LIN {X 0,Y 546.313,Z 765.202,A -85,B 0,C 180,E1 25447.625,E2 25447.625} C_VEL
LIN {X 0,Y 547.105,Z 747.49,A -85,B 0,C 180,E1 25445.835,E2 25445.835} C_VEL
LIN {X 0,Y 547.912,Z 730.024,A -85,B 0,C 180,E1 25444.317,E2 25444.317} C_VEL
LIN {X 0,Y 548.795,Z 710.07,A -85,B 0,C 180,E1 25442.846,E2 25442.846} C_VEL
LIN {X 0,Y 549.579,Z 691.702,A -85,B 0,C 180,E1 25441.708,E2 25441.708} C_VEL
LIN {X 0,Y 550.398,Z 670.915,A -85,B 0,C 180,E1 25440.628,E2 25440.628} C_VEL
LIN {X 0,Y 551.103,Z 650.987,A -85,B 0,C 180,E1 25439.802,E2 25439.802} C_VEL
LIN {X 0,Y 551.691,Z 629.673,A -85,B 0,C 180,E1 25439.106,E2 25439.106} C_VEL
LIN {X 0,Y 552.189,Z 607.333,A -85,B 0,C 180,E1 25438.596,E2 25438.596} C_VEL
LIN {X 0,Y 553.481,Z 453.484,A -85,B 0,C 180,E1 25436.326,E2 25436.326} C_VEL
LIN {X 0,Y 554.426,Z 320.88,A -85,B 0,C 180,E1 25434.346,E2 25434.346} C_VEL
LIN {X 0,Y 549.959,Z 305.52,A -85,B 0,C 180,E1 25433.742,E2 25433.742} C_VEL
LIN {X 0,Y 550.398,Z 290.694,A -85,B 0,C 180,E1 25431.989,E2 25431.989} C_VEL
LIN {X 0,Y 545.865,Z 277.355,A -85,B 0,C 180,E1 25429.964,E2 25429.964} C_VEL
LIN {X 0,Y 544.39,Z 272.482,A -85,B 0,C 180,E1 25429.174,E2 25429.174} C_VEL
LIN {X 0,Y 544.34,Z 272.43,A -85,B 0,C 180,E1 25426.028,E2 25426.028} C_VEL
LIN {X 0,Y 544.339,Z 272.424,A -85,B 0,C 180,E1 25422.562,E2 25422.562} C_VEL
LIN {X 0,Y 544.397,Z 272.403,A -85,B 0,C 180,E1 25419.358,E2 25419.358} C_VEL
LIN {X 0,Y 544.337,Z 272.425,A -85,B 0,C 180,E1 25416.081,E2 25416.081} C_VEL
LIN {X 0,Y 544.365,Z 272.425,A -85,B 0,C 180,E1 25412.733,E2 25412.733} C_VEL
LIN {X 0,Y 544.362,Z 272.42,A -85,B 0,C 180,E1 25409.609,E2 25409.609} C_VEL
LIN {X 0,Y 544.344,Z 272.417,A -85,B 0,C 180,E1 25406.274,E2 25406.274} C_VEL
LIN {X 0,Y 544.409,Z 272.422,A -85,B 0,C 180,E1 25403.029,E2 25403.029} C_VEL
LIN {X 0,Y 544.349,Z 272.415,A -85,B 0,C 180,E1 25399.753,E2 25399.753} C_VEL
LIN {X 0,Y 544.358,Z 272.418,A -85,B 0,C 180,E1 25396.321,E2 25396.321} C_VEL
LIN {X 0,Y 544.4,Z 272.421,A -85,B 0,C 180,E1 25393.056,E2 25393.056} C_VEL
LIN {X 0,Y 544.35,Z 272.418,A -85,B 0,C 180,E1 25389.729,E2 25389.729} C_VEL
LIN {X 0,Y 544.384,Z 272.422,A -85,B 0,C 180,E1 25386.433,E2 25386.433} C_VEL
LIN {X 0,Y 544.382,Z 272.416,A -85,B 0,C 180,E1 25383.159,E2 25383.159} C_VEL
LIN {X 0,Y 544.354,Z 272.423,A -85,B 0,C 180,E1 25379.79,E2 25379.79} C_VEL
LIN {X 0,Y 544.402,Z 272.411,A -85,B 0,C 180,E1 25376.525,E2 25376.525} C_VEL
LIN {X 0,Y 544.369,Z 272.425,A -85,B 0,C 180,E1 25373.249,E2 25373.249} C_VEL
LIN {X 0,Y 544.364,Z 272.413,A -85,B 0,C 180,E1 25369.844,E2 25369.844} C_VEL
LIN {X 0,Y 544.406,Z 272.418,A -85,B 0,C 180,E1 25366.512,E2 25366.512} C_VEL
LIN {X 0,Y 544.366,Z 272.417,A -85,B 0,C 180,E1 25363.24,E2 25363.24} C_VEL
LIN {X 0,Y 544.374,Z 272.42,A -85,B 0,C 180,E1 25359.8,E2 25359.8} C_VEL
LIN {X 0,Y 544.406,Z 272.424,A -85,B 0,C 180,E1 25356.513,E2 25356.513} C_VEL
LIN {X 0,Y 544.37,Z 272.424,A -85,B 0,C 180,E1 25353.139,E2 25353.139} C_VEL
LIN {X 0,Y 544.378,Z 272.421,A -85,B 0,C 180,E1 25349.663,E2 25349.663} C_VEL
LIN {X 0,Y 544.374,Z 272.425,A -85,B 0,C 180,E1 25349.04,E2 25349.04} C_VEL
LIN {X 0,Y 543.409,Z 272.55,A -85,B 0,C 180,E1 25348.229,E2 25348.229} C_VEL
LIN {X 0,Y 536.878,Z 273.358,A -85,B 0,C 180,E1 25345.892,E2 25345.892} C_VEL
LIN {X 0,Y 536.432,Z 273.411,A -85,B 0,C 180,E1 25345.358,E2 25345.358} C_VEL
LIN {X 0,Y 536.464,Z 273.409,A -85,B 0,C 180,E1 25342.033,E2 25342.033} C_VEL
LIN {X 0,Y 536.459,Z 273.413,A -85,B 0,C 180,E1 25338.574,E2 25338.574} C_VEL
LIN {X 0,Y 536.436,Z 273.411,A -85,B 0,C 180,E1 25335.207,E2 25335.207} C_VEL
LIN {X 0,Y 536.465,Z 273.408,A -85,B 0,C 180,E1 25331.797,E2 25331.797} C_VEL
LIN {X 0,Y 536.465,Z 273.414,A -85,B 0,C 180,E1 25328.311,E2 25328.311} C_VEL
LIN {X 0,Y 536.441,Z 273.412,A -85,B 0,C 180,E1 25324.903,E2 25324.903} C_VEL
LIN {X 0,Y 536.461,Z 273.407,A -85,B 0,C 180,E1 25321.456,E2 25321.456} C_VEL
LIN {X 0,Y 536.459,Z 273.411,A -85,B 0,C 180,E1 25318.013,E2 25318.013} C_VEL
LIN {X 0,Y 536.444,Z 273.411,A -85,B 0,C 180,E1 25314.676,E2 25314.676} C_VEL
LIN {X 0,Y 536.457,Z 273.407,A -85,B 0,C 180,E1 25311.197,E2 25311.197} C_VEL
LIN {X 0,Y 536.456,Z 273.411,A -85,B 0,C 180,E1 25307.747,E2 25307.747} C_VEL
LIN {X 0,Y 536.455,Z 273.415,A -85,B 0,C 180,E1 25304.352,E2 25304.352} C_VEL
LIN {X 0,Y 536.45,Z 273.41,A -85,B 0,C 180,E1 25300.85,E2 25300.85} C_VEL
LIN {X 0,Y 536.452,Z 273.41,A -85,B 0,C 180,E1 25297.45,E2 25297.45} C_VEL
LIN {X 0,Y 536.46,Z 273.414,A -85,B 0,C 180,E1 25294.061,E2 25294.061} C_VEL
LIN {X 0,Y 536.451,Z 273.409,A -85,B 0,C 180,E1 25290.641,E2 25290.641} C_VEL
LIN {X 0,Y 536.453,Z 273.408,A -85,B 0,C 180,E1 25287.222,E2 25287.222} C_VEL
LIN {X 0,Y 536.458,Z 273.413,A -85,B 0,C 180,E1 25283.794,E2 25283.794} C_VEL
LIN {X 0,Y 536.453,Z 273.412,A -85,B 0,C 180,E1 25280.344,E2 25280.344} C_VEL
LIN {X 0,Y 536.457,Z 273.408,A -85,B 0,C 180,E1 25276.967,E2 25276.967} C_VEL
LIN {X 0,Y 536.451,Z 273.414,A -85,B 0,C 180,E1 25273.543,E2 25273.543} C_VEL
LIN {X 0,Y 536.456,Z 273.412,A -85,B 0,C 180,E1 25270.171,E2 25270.171} C_VEL
LIN {X 0,Y 536.458,Z 273.407,A -85,B 0,C 180,E1 25266.727,E2 25266.727} C_VEL
LIN {X 0,Y 536.444,Z 273.411,A -85,B 0,C 180,E1 25263.309,E2 25263.309} C_VEL
LIN {X 0,Y 536.461,Z 273.412,A -85,B 0,C 180,E1 25259.911,E2 25259.911} C_VEL
LIN {X 0,Y 536.462,Z 273.407,A -85,B 0,C 180,E1 25256.42,E2 25256.42} C_VEL
LIN {X 0,Y 536.438,Z 273.411,A -85,B 0,C 180,E1 25252.985,E2 25252.985} C_VEL
LIN {X 0,Y 536.463,Z 273.413,A -85,B 0,C 180,E1 25249.565,E2 25249.565} C_VEL
LIN {X 0,Y 536.463,Z 273.409,A -85,B 0,C 180,E1 25246.107,E2 25246.107} C_VEL
LIN {X 0,Y 536.436,Z 273.411,A -85,B 0,C 180,E1 25242.723,E2 25242.723} C_VEL
LIN {X 0,Y 536.456,Z 273.414,A -85,B 0,C 180,E1 25239.323,E2 25239.323} C_VEL
LIN {X 0,Y 536.465,Z 273.409,A -85,B 0,C 180,E1 25235.951,E2 25235.951} C_VEL
LIN {X 0,Y 536.431,Z 273.411,A -85,B 0,C 180,E1 25232.593,E2 25232.593} C_VEL
LIN {X 0,Y 536.454,Z 273.415,A -85,B 0,C 180,E1 25229.23,E2 25229.23} C_VEL
LIN {X 0,Y 536.464,Z 273.409,A -85,B 0,C 180,E1 25225.817,E2 25225.817} C_VEL
LIN {X 0,Y 536.427,Z 273.412,A -85,B 0,C 180,E1 25222.464,E2 25222.464} C_VEL
LIN {X 0,Y 536.445,Z 273.415,A -85,B 0,C 180,E1 25219.037,E2 25219.037} C_VEL
LIN {X 0,Y 536.465,Z 273.4,A -85,B 0,C 180,E1 25215.679,E2 25215.679} C_VEL
LIN {X 0,Y 536.421,Z 273.412,A -85,B 0,C 180,E1 25212.378,E2 25212.378} C_VEL
LIN {X 0,Y 536.444,Z 273.405,A -85,B 0,C 180,E1 25208.952,E2 25208.952} C_VEL
LIN {X 0,Y 536.462,Z 273.41,A -85,B 0,C 180,E1 25205.562,E2 25205.562} C_VEL
LIN {X 0,Y 536.416,Z 273.407,A -85,B 0,C 180,E1 25202.243,E2 25202.243} C_VEL
LIN {X 0,Y 536.45,Z 273.408,A -85,B 0,C 180,E1 25198.932,E2 25198.932} C_VEL
LIN {X 0,Y 536.442,Z 273.404,A -85,B 0,C 180,E1 25195.617,E2 25195.617} C_VEL
LIN {X 0,Y 536.413,Z 273.406,A -85,B 0,C 180,E1 25192.287,E2 25192.287} C_VEL
LIN {X 0,Y 536.459,Z 273.411,A -85,B 0,C 180,E1 25188.932,E2 25188.932} C_VEL
LIN {X 0,Y 536.425,Z 273.404,A -85,B 0,C 180,E1 25185.647,E2 25185.647} C_VEL
LIN {X 0,Y 536.412,Z 273.414,A -85,B 0,C 180,E1 25182.263,E2 25182.263} C_VEL
LIN {X 0,Y 536.467,Z 273.399,A -85,B 0,C 180,E1 25179.024,E2 25179.024} C_VEL
LIN {X 0,Y 536.406,Z 273.412,A -85,B 0,C 180,E1 25175.79,E2 25175.79} C_VEL
LIN {X 0,Y 536.419,Z 273.416,A -85,B 0,C 180,E1 25172.347,E2 25172.347} C_VEL
LIN {X 0,Y 536.44,Z 273.406,A -85,B 0,C 180,E1 25169.165,E2 25169.165} C_VEL
LIN {X 0,Y 536.4,Z 273.412,A -85,B 0,C 180,E1 25165.853,E2 25165.853} C_VEL
LIN {X 0,Y 536.446,Z 273.394,A -85,B 0,C 180,E1 25162.559,E2 25162.559} C_VEL
LIN {X 0,Y 536.408,Z 273.414,A -85,B 0,C 180,E1 25159.343,E2 25159.343} C_VEL
LIN {X 0,Y 536.397,Z 273.394,A -85,B 0,C 180,E1 25155.951,E2 25155.951} C_VEL
LIN {X 0,Y 536.455,Z 273.391,A -85,B 0,C 180,E1 25152.72,E2 25152.72} C_VEL
LIN {X 0,Y 536.44,Z 273.685,A -85,B 0,C 180,E1 25151.314,E2 25151.314} C_VEL
LIN {X 0,Y 542.981,Z 293.04,A -85,B 0,C 180,E1 25148.331,E2 25148.331} C_VEL
LIN {X 0,Y 543.254,Z 295.295,A -85,B 0,C 180,E1 25148.026,E2 25148.026} C_VEL
LIN {X 0,Y 542.934,Z 306,A -85,B 0,C 180,E1 25146.777,E2 25146.777} C_VEL
LIN {X 0,Y 548.053,Z 324.047,A -85,B 0,C 180,E1 25146.083,E2 25146.083} C_VEL
LIN {X 0,Y 546.001,Z 542.335,A -85,B 0,C 180,E1 25142.826,E2 25142.826} C_VEL
LIN {X 0,Y 545.341,Z 608.353,A -85,B 0,C 180,E1 25141.825,E2 25141.825} C_VEL
LIN {X 0,Y 544.737,Z 631.517,A -85,B 0,C 180,E1 25141.275,E2 25141.275} C_VEL
LIN {X 0,Y 544.078,Z 652.53,A -85,B 0,C 180,E1 25140.569,E2 25140.569} C_VEL
LIN {X 0,Y 543.247,Z 673.374,A -85,B 0,C 180,E1 25139.675,E2 25139.675} C_VEL
LIN {X 0,Y 542.36,Z 692.723,A -85,B 0,C 180,E1 25138.64,E2 25138.64} C_VEL
LIN {X 0,Y 541.446,Z 711.788,A -85,B 0,C 180,E1 25137.434,E2 25137.434} C_VEL
LIN {X 0,Y 540.442,Z 731.276,A -85,B 0,C 180,E1 25135.955,E2 25135.955} C_VEL
LIN {X 0,Y 539.566,Z 748.034,A -85,B 0,C 180,E1 25134.472,E2 25134.472} C_VEL
LIN {X 0,Y 538.636,Z 766.218,A -85,B 0,C 180,E1 25132.596,E2 25132.596} C_VEL
LIN {X 0,Y 537.875,Z 782.057,A -85,B 0,C 180,E1 25130.682,E2 25130.682} C_VEL
LIN {X 0,Y 537.22,Z 797.018,A -85,B 0,C 180,E1 25128.557,E2 25128.557} C_VEL
LIN {X 0,Y 536.79,Z 808.45,A -85,B 0,C 180,E1 25126.669,E2 25126.669} C_VEL
LIN {X 0,Y 536.423,Z 819.843,A -85,B 0,C 180,E1 25124.463,E2 25124.463} C_VEL
LIN {X 0,Y 536.179,Z 829.242,A -85,B 0,C 180,E1 25122.274,E2 25122.274} C_VEL
LIN {X 0,Y 536.037,Z 836.893,A -85,B 0,C 180,E1 25120.098,E2 25120.098} C_VEL
LIN {X 0,Y 535.954,Z 843.407,A -85,B 0,C 180,E1 25117.719,E2 25117.719} C_VEL
LIN {X 0,Y 535.926,Z 847.982,A -85,B 0,C 180,E1 25115.46,E2 25115.46} C_VEL
LIN {X 0,Y 535.914,Z 851.142,A -85,B 0,C 180,E1 25112.994,E2 25112.994} C_VEL
LIN {X 0,Y 535.902,Z 852.351,A -85,B 0,C 180,E1 25110.748,E2 25110.748} C_VEL
LIN {X 0,Y 535.898,Z 852.161,A -85,B 0,C 180,E1 25108.503,E2 25108.503} C_VEL
LIN {X 0,Y 535.907,Z 850.245,A -85,B 0,C 180,E1 25106.149,E2 25106.149} C_VEL
LIN {X 0,Y 535.926,Z 846.625,A -85,B 0,C 180,E1 25103.788,E2 25103.788} C_VEL
LIN {X 0,Y 535.966,Z 841.189,A -85,B 0,C 180,E1 25101.388,E2 25101.388} C_VEL
LIN {X 0,Y 536.063,Z 834.754,A -85,B 0,C 180,E1 25099.251,E2 25099.251} C_VEL
LIN {X 0,Y 536.246,Z 826.17,A -85,B 0,C 180,E1 25096.962,E2 25096.962} C_VEL
LIN {X 0,Y 536.526,Z 816.092,A -85,B 0,C 180,E1 25094.766,E2 25094.766} C_VEL
LIN {X 0,Y 536.92,Z 804.629,A -85,B 0,C 180,E1 25092.666,E2 25092.666} C_VEL
LIN {X 0,Y 537.476,Z 791.027,A -85,B 0,C 180,E1 25090.55,E2 25090.55} C_VEL
LIN {X 0,Y 538.165,Z 776.094,A -85,B 0,C 180,E1 25088.561,E2 25088.561} C_VEL
LIN {X 0,Y 538.977,Z 759.485,A -85,B 0,C 180,E1 25086.675,E2 25086.675} C_VEL
LIN {X 0,Y 539.771,Z 743.826,A -85,B 0,C 180,E1 25085.135,E2 25085.135} C_VEL
LIN {X 0,Y 540.769,Z 725.001,A -85,B 0,C 180,E1 25083.539,E2 25083.539} C_VEL
LIN {X 0,Y 541.748,Z 705.74,A -85,B 0,C 180,E1 25082.165,E2 25082.165} C_VEL
LIN {X 0,Y 542.698,Z 685.746,A -85,B 0,C 180,E1 25080.958,E2 25080.958} C_VEL
LIN {X 0,Y 543.551,Z 665.758,A -85,B 0,C 180,E1 25079.978,E2 25079.978} C_VEL
LIN {X 0,Y 544.316,Z 645.503,A -85,B 0,C 180,E1 25079.171,E2 25079.171} C_VEL
LIN {X 0,Y 544.997,Z 622.893,A -85,B 0,C 180,E1 25078.495,E2 25078.495} C_VEL
LIN {X 0,Y 545.412,Z 602.857,A -85,B 0,C 180,E1 25078.077,E2 25078.077} C_VEL
LIN {X 0,Y 547.508,Z 380.748,A -85,B 0,C 180,E1 25074.772,E2 25074.772} C_VEL
LIN {X 0,Y 547.876,Z 322.729,A -85,B 0,C 180,E1 25073.882,E2 25073.882} C_VEL
LIN {X 0,Y 542.859,Z 305.414,A -85,B 0,C 180,E1 25073.182,E2 25073.182} C_VEL
LIN {X 0,Y 543.113,Z 293.49,A -85,B 0,C 180,E1 25071.737,E2 25071.737} C_VEL
LIN {X 0,Y 537.234,Z 276.036,A -85,B 0,C 180,E1 25069.073,E2 25069.073} C_VEL
LIN {X 0,Y 536.41,Z 273.513,A -85,B 0,C 180,E1 25068.624,E2 25068.624} C_VEL
LIN {X 0,Y 536.458,Z 273.405,A -85,B 0,C 180,E1 25065.361,E2 25065.361} C_VEL
LIN {X 0,Y 536.397,Z 273.414,A -85,B 0,C 180,E1 25062.11,E2 25062.11} C_VEL
LIN {X 0,Y 536.417,Z 273.388,A -85,B 0,C 180,E1 25058.777,E2 25058.777} C_VEL
LIN {X 0,Y 536.434,Z 273.415,A -85,B 0,C 180,E1 25055.559,E2 25055.559} C_VEL
LIN {X 0,Y 536.4,Z 273.415,A -85,B 0,C 180,E1 25052.195,E2 25052.195} C_VEL
LIN {X 0,Y 536.46,Z 273.413,A -85,B 0,C 180,E1 25048.986,E2 25048.986} C_VEL
LIN {X 0,Y 536.412,Z 273.406,A -85,B 0,C 180,E1 25045.741,E2 25045.741} C_VEL
LIN {X 0,Y 536.412,Z 273.411,A -85,B 0,C 180,E1 25042.349,E2 25042.349} C_VEL
LIN {X 0,Y 536.463,Z 273.406,A -85,B 0,C 180,E1 25039.105,E2 25039.105} C_VEL
LIN {X 0,Y 536.409,Z 273.408,A -85,B 0,C 180,E1 25035.792,E2 25035.792} C_VEL
LIN {X 0,Y 536.43,Z 273.411,A -85,B 0,C 180,E1 25032.377,E2 25032.377} C_VEL
LIN {X 0,Y 536.452,Z 273.401,A -85,B 0,C 180,E1 25029.116,E2 25029.116} C_VEL
LIN {X 0,Y 536.414,Z 273.413,A -85,B 0,C 180,E1 25025.777,E2 25025.777} C_VEL
LIN {X 0,Y 536.453,Z 273.401,A -85,B 0,C 180,E1 25022.457,E2 25022.457} C_VEL
LIN {X 0,Y 536.442,Z 273.415,A -85,B 0,C 180,E1 25019.146,E2 25019.146} C_VEL
LIN {X 0,Y 536.416,Z 273.403,A -85,B 0,C 180,E1 25015.724,E2 25015.724} C_VEL
LIN {X 0,Y 536.466,Z 273.405,A -85,B 0,C 180,E1 25012.396,E2 25012.396} C_VEL
LIN {X 0,Y 536.442,Z 273.405,A -85,B 0,C 180,E1 25009.041,E2 25009.041} C_VEL
LIN {X 0,Y 536.423,Z 273.407,A -85,B 0,C 180,E1 25005.647,E2 25005.647} C_VEL
LIN {X 0,Y 536.464,Z 273.41,A -85,B 0,C 180,E1 25002.314,E2 25002.314} C_VEL
LIN {X 0,Y 536.447,Z 273.415,A -85,B 0,C 180,E1 24998.917,E2 24998.917} C_VEL
LIN {X 0,Y 536.43,Z 273.411,A -85,B 0,C 180,E1 24995.557,E2 24995.557} C_VEL
LIN {X 0,Y 536.465,Z 273.41,A -85,B 0,C 180,E1 24992.229,E2 24992.229} C_VEL
LIN {X 0,Y 536.45,Z 273.415,A -85,B 0,C 180,E1 24988.792,E2 24988.792} C_VEL
LIN {X 0,Y 536.432,Z 273.411,A -85,B 0,C 180,E1 24985.358,E2 24985.358} C_VEL
LIN {X 0,Y 535.448,Z 273.54,A -85,B 0,C 180,E1 24984.535,E2 24984.535} C_VEL
LIN {X 0,Y 528.972,Z 274.344,A -85,B 0,C 180,E1 24982.164,E2 24982.164} C_VEL
LIN {X 0,Y 528.508,Z 274.398,A -85,B 0,C 180,E1 24981.622,E2 24981.622} C_VEL
LIN {X 0,Y 528.524,Z 274.401,A -85,B 0,C 180,E1 24978.189,E2 24978.189} C_VEL
LIN {X 0,Y 528.509,Z 274.403,A -85,B 0,C 180,E1 24974.728,E2 24974.728} C_VEL
LIN {X 0,Y 528.504,Z 274.399,A -85,B 0,C 180,E1 24971.317,E2 24971.317} C_VEL
LIN {X 0,Y 528.522,Z 274.399,A -85,B 0,C 180,E1 24967.919,E2 24967.919} C_VEL
LIN {X 0,Y 528.517,Z 274.402,A -85,B 0,C 180,E1 24964.429,E2 24964.429} C_VEL
LIN {X 0,Y 528.502,Z 274.399,A -85,B 0,C 180,E1 24960.969,E2 24960.969} C_VEL
LIN {X 0,Y 528.523,Z 274.395,A -85,B 0,C 180,E1 24957.612,E2 24957.612} C_VEL
LIN {X 0,Y 528.522,Z 274.402,A -85,B 0,C 180,E1 24954.118,E2 24954.118} C_VEL
LIN {X 0,Y 528.505,Z 274.401,A -85,B 0,C 180,E1 24950.718,E2 24950.718} C_VEL
LIN {X 0,Y 528.522,Z 274.397,A -85,B 0,C 180,E1 24947.278,E2 24947.278} C_VEL
LIN {X 0,Y 528.516,Z 274.402,A -85,B 0,C 180,E1 24943.79,E2 24943.79} C_VEL
LIN {X 0,Y 528.514,Z 274.402,A -85,B 0,C 180,E1 24940.344,E2 24940.344} C_VEL
LIN {X 0,Y 528.515,Z 274.398,A -85,B 0,C 180,E1 24936.845,E2 24936.845} C_VEL
LIN {X 0,Y 528.513,Z 274.399,A -85,B 0,C 180,E1 24933.471,E2 24933.471} C_VEL
LIN {X 0,Y 528.525,Z 274.404,A -85,B 0,C 180,E1 24930,E2 24930} C_VEL
LIN {X 0,Y 528.513,Z 274.399,A -85,B 0,C 180,E1 24926.529,E2 24926.529} C_VEL
LIN {X 0,Y 528.521,Z 274.397,A -85,B 0,C 180,E1 24923.046,E2 24923.046} C_VEL
LIN {X 0,Y 528.51,Z 274.403,A -85,B 0,C 180,E1 24919.536,E2 24919.536} C_VEL
LIN {X 0,Y 528.518,Z 274.402,A -85,B 0,C 180,E1 24916.098,E2 24916.098} C_VEL
LIN {X 0,Y 528.523,Z 274.397,A -85,B 0,C 180,E1 24912.609,E2 24912.609} C_VEL
LIN {X 0,Y 528.506,Z 274.399,A -85,B 0,C 180,E1 24909.16,E2 24909.16} C_VEL
LIN {X 0,Y 528.523,Z 274.403,A -85,B 0,C 180,E1 24905.761,E2 24905.761} C_VEL
LIN {X 0,Y 528.52,Z 274.397,A -85,B 0,C 180,E1 24902.266,E2 24902.266} C_VEL
LIN {X 0,Y 528.504,Z 274.398,A -85,B 0,C 180,E1 24898.905,E2 24898.905} C_VEL
LIN {X 0,Y 528.51,Z 274.402,A -85,B 0,C 180,E1 24895.381,E2 24895.381} C_VEL
LIN {X 0,Y 528.523,Z 274.401,A -85,B 0,C 180,E1 24891.924,E2 24891.924} C_VEL
LIN {X 0,Y 528.513,Z 274.398,A -85,B 0,C 180,E1 24888.518,E2 24888.518} C_VEL
LIN {X 0,Y 528.499,Z 274.402,A -85,B 0,C 180,E1 24885.037,E2 24885.037} C_VEL
LIN {X 0,Y 528.524,Z 274.402,A -85,B 0,C 180,E1 24881.607,E2 24881.607} C_VEL
LIN {X 0,Y 528.527,Z 274.397,A -85,B 0,C 180,E1 24878.098,E2 24878.098} C_VEL
LIN {X 0,Y 528.492,Z 274.401,A -85,B 0,C 180,E1 24874.713,E2 24874.713} C_VEL
LIN {X 0,Y 528.522,Z 274.402,A -85,B 0,C 180,E1 24871.349,E2 24871.349} C_VEL
LIN {X 0,Y 528.527,Z 274.398,A -85,B 0,C 180,E1 24867.857,E2 24867.857} C_VEL
LIN {X 0,Y 528.491,Z 274.4,A -85,B 0,C 180,E1 24864.477,E2 24864.477} C_VEL
LIN {X 0,Y 528.507,Z 274.404,A -85,B 0,C 180,E1 24861.066,E2 24861.066} C_VEL
LIN {X 0,Y 528.526,Z 274.4,A -85,B 0,C 180,E1 24857.619,E2 24857.619} C_VEL
LIN {X 0,Y 528.488,Z 274.395,A -85,B 0,C 180,E1 24854.238,E2 24854.238} C_VEL
LIN {X 0,Y 528.492,Z 274.392,A -85,B 0,C 180,E1 24850.795,E2 24850.795} C_VEL
LIN {X 0,Y 528.528,Z 274.396,A -85,B 0,C 180,E1 24847.391,E2 24847.391} C_VEL
LIN {X 0,Y 528.487,Z 274.39,A -85,B 0,C 180,E1 24844.014,E2 24844.014} C_VEL
LIN {X 0,Y 528.483,Z 274.403,A -85,B 0,C 180,E1 24840.542,E2 24840.542} C_VEL
LIN {X 0,Y 528.525,Z 274.386,A -85,B 0,C 180,E1 24837.181,E2 24837.181} C_VEL
LIN {X 0,Y 528.486,Z 274.401,A -85,B 0,C 180,E1 24833.809,E2 24833.809} C_VEL
LIN {X 0,Y 528.478,Z 274.396,A -85,B 0,C 180,E1 24830.416,E2 24830.416} C_VEL
LIN {X 0,Y 528.527,Z 274.401,A -85,B 0,C 180,E1 24827.101,E2 24827.101} C_VEL
LIN {X 0,Y 528.473,Z 274.397,A -85,B 0,C 180,E1 24823.852,E2 24823.852} C_VEL
LIN {X 0,Y 528.481,Z 274.393,A -85,B 0,C 180,E1 24820.418,E2 24820.418} C_VEL
LIN {X 0,Y 528.529,Z 274.399,A -85,B 0,C 180,E1 24817.064,E2 24817.064} C_VEL
LIN {X 0,Y 528.468,Z 274.394,A -85,B 0,C 180,E1 24813.722,E2 24813.722} C_VEL
LIN {X 0,Y 528.475,Z 274.397,A -85,B 0,C 180,E1 24810.272,E2 24810.272} C_VEL
LIN {X 0,Y 528.515,Z 274.401,A -85,B 0,C 180,E1 24806.986,E2 24806.986} C_VEL
LIN {X 0,Y 528.46,Z 274.403,A -85,B 0,C 180,E1 24803.687,E2 24803.687} C_VEL
LIN {X 0,Y 528.486,Z 274.384,A -85,B 0,C 180,E1 24800.353,E2 24800.353} C_VEL
LIN {X 0,Y 528.474,Z 274.391,A -85,B 0,C 180,E1 24797.218,E2 24797.218} C_VEL
LIN {X 0,Y 528.458,Z 274.409,A -85,B 0,C 180,E1 24793.825,E2 24793.825} C_VEL
LIN {X 0,Y 528.482,Z 274.553,A -85,B 0,C 180,E1 24791.93,E2 24791.93} C_VEL
LIN {X 0,Y 534.575,Z 292.474,A -85,B 0,C 180,E1 24789.072,E2 24789.072} C_VEL
LIN {X 0,Y 536.088,Z 297.512,A -85,B 0,C 180,E1 24788.326,E2 24788.326} C_VEL
LIN {X 0,Y 535.857,Z 305.967,A -85,B 0,C 180,E1 24787.343,E2 24787.343} C_VEL
LIN {X 0,Y 541.567,Z 325.996,A -85,B 0,C 180,E1 24786.554,E2 24786.554} C_VEL
LIN {X 0,Y 539.267,Z 543.699,A -85,B 0,C 180,E1 24783.267,E2 24783.267} C_VEL
LIN {X 0,Y 538.539,Z 608.332,A -85,B 0,C 180,E1 24782.276,E2 24782.276} C_VEL
LIN {X 0,Y 537.871,Z 631.493,A -85,B 0,C 180,E1 24781.72,E2 24781.72} C_VEL
LIN {X 0,Y 537.162,Z 651.73,A -85,B 0,C 180,E1 24781.037,E2 24781.037} C_VEL
LIN {X 0,Y 536.269,Z 672.198,A -85,B 0,C 180,E1 24780.163,E2 24780.163} C_VEL
LIN {X 0,Y 535.262,Z 691.734,A -85,B 0,C 180,E1 24779.117,E2 24779.117} C_VEL
LIN {X 0,Y 534.288,Z 709.997,A -85,B 0,C 180,E1 24777.958,E2 24777.958} C_VEL
LIN {X 0,Y 533.143,Z 730.006,A -85,B 0,C 180,E1 24776.449,E2 24776.449} C_VEL
LIN {X 0,Y 532.113,Z 747.103,A -85,B 0,C 180,E1 24774.928,E2 24774.928} C_VEL
LIN {X 0,Y 531.084,Z 765.208,A -85,B 0,C 180,E1 24773.053,E2 24773.053} C_VEL
LIN {X 0,Y 530.256,Z 780.297,A -85,B 0,C 180,E1 24771.225,E2 24771.225} C_VEL
LIN {X 0,Y 529.53,Z 794.888,A -85,B 0,C 180,E1 24769.18,E2 24769.18} C_VEL
LIN {X 0,Y 528.965,Z 807.183,A -85,B 0,C 180,E1 24767.149,E2 24767.149} C_VEL
LIN {X 0,Y 528.531,Z 818.808,A -85,B 0,C 180,E1 24764.908,E2 24764.908} C_VEL
LIN {X 0,Y 528.242,Z 828.386,A -85,B 0,C 180,E1 24762.683,E2 24762.683} C_VEL
LIN {X 0,Y 528.074,Z 835.83,A -85,B 0,C 180,E1 24760.583,E2 24760.583} C_VEL
LIN {X 0,Y 527.977,Z 842.646,A -85,B 0,C 180,E1 24758.165,E2 24758.165} C_VEL
LIN {X 0,Y 527.926,Z 847.218,A -85,B 0,C 180,E1 24755.979,E2 24755.979} C_VEL
LIN {X 0,Y 527.905,Z 850.476,A -85,B 0,C 180,E1 24753.692,E2 24753.692} C_VEL
LIN {X 0,Y 527.905,Z 852.218,A -85,B 0,C 180,E1 24751.302,E2 24751.302} C_VEL
LIN {X 0,Y 527.907,Z 852.325,A -85,B 0,C 180,E1 24749.132,E2 24749.132} C_VEL
LIN {X 0,Y 527.917,Z 850.925,A -85,B 0,C 180,E1 24746.743,E2 24746.743} C_VEL
LIN {X 0,Y 527.926,Z 847.788,A -85,B 0,C 180,E1 24744.348,E2 24744.348} C_VEL
LIN {X 0,Y 527.965,Z 843.408,A -85,B 0,C 180,E1 24742.163,E2 24742.163} C_VEL
LIN {X 0,Y 528.062,Z 836.894,A -85,B 0,C 180,E1 24739.748,E2 24739.748} C_VEL
LIN {X 0,Y 528.223,Z 829.237,A -85,B 0,C 180,E1 24737.539,E2 24737.539} C_VEL
LIN {X 0,Y 528.502,Z 819.847,A -85,B 0,C 180,E1 24735.315,E2 24735.315} C_VEL
LIN {X 0,Y 528.928,Z 808.252,A -85,B 0,C 180,E1 24733.041,E2 24733.041} C_VEL
LIN {X 0,Y 529.451,Z 796.307,A -85,B 0,C 180,E1 24731.046,E2 24731.046} C_VEL
LIN {X 0,Y 530.209,Z 781.182,A -85,B 0,C 180,E1 24728.889,E2 24728.889} C_VEL
LIN {X 0,Y 531.04,Z 765.933,A -85,B 0,C 180,E1 24727.029,E2 24727.029} C_VEL
LIN {X 0,Y 532.093,Z 747.489,A -85,B 0,C 180,E1 24725.108,E2 24725.108} C_VEL
LIN {X 0,Y 533.099,Z 730.689,A -85,B 0,C 180,E1 24723.609,E2 24723.609} C_VEL
LIN {X 0,Y 534.238,Z 710.915,A -85,B 0,C 180,E1 24722.103,E2 24722.103} C_VEL
LIN {X 0,Y 535.212,Z 692.716,A -85,B 0,C 180,E1 24720.941,E2 24720.941} C_VEL
LIN {X 0,Y 536.202,Z 673.368,A -85,B 0,C 180,E1 24719.895,E2 24719.895} C_VEL
LIN {X 0,Y 537.134,Z 652.511,A -85,B 0,C 180,E1 24718.993,E2 24718.993} C_VEL
LIN {X 0,Y 537.852,Z 631.97,A -85,B 0,C 180,E1 24718.294,E2 24718.294} C_VEL
LIN {X 0,Y 538.536,Z 608.644,A -85,B 0,C 180,E1 24717.73,E2 24717.73} C_VEL
LIN {X 0,Y 539.216,Z 548.569,A -85,B 0,C 180,E1 24716.805,E2 24716.805} C_VEL
LIN {X 0,Y 541.486,Z 333.024,A -85,B 0,C 180,E1 24713.554,E2 24713.554} C_VEL
LIN {X 0,Y 541.381,Z 324.653,A -85,B 0,C 180,E1 24713.41,E2 24713.41} C_VEL
LIN {X 0,Y 535.792,Z 305.405,A -85,B 0,C 180,E1 24712.615,E2 24712.615} C_VEL
LIN {X 0,Y 535.979,Z 296.835,A -85,B 0,C 180,E1 24711.582,E2 24711.582} C_VEL
LIN {X 0,Y 529.435,Z 277.413,A -85,B 0,C 180,E1 24708.568,E2 24708.568} C_VEL
LIN {X 0,Y 528.476,Z 274.5,A -85,B 0,C 180,E1 24708.034,E2 24708.034} C_VEL
LIN {X 0,Y 528.458,Z 274.384,A -85,B 0,C 180,E1 24704.583,E2 24704.583} C_VEL
LIN {X 0,Y 528.526,Z 274.404,A -85,B 0,C 180,E1 24701.318,E2 24701.318} C_VEL
LIN {X 0,Y 528.458,Z 274.379,A -85,B 0,C 180,E1 24698.083,E2 24698.083} C_VEL
LIN {X 0,Y 528.483,Z 274.4,A -85,B 0,C 180,E1 24694.713,E2 24694.713} C_VEL
LIN {X 0,Y 528.502,Z 274.405,A -85,B 0,C 180,E1 24691.437,E2 24691.437} C_VEL
LIN {X 0,Y 528.463,Z 274.404,A -85,B 0,C 180,E1 24688.106,E2 24688.106} C_VEL
LIN {X 0,Y 528.506,Z 274.399,A -85,B 0,C 180,E1 24684.76,E2 24684.76} C_VEL
LIN {X 0,Y 528.484,Z 274.399,A -85,B 0,C 180,E1 24681.533,E2 24681.533} C_VEL
LIN {X 0,Y 528.473,Z 274.401,A -85,B 0,C 180,E1 24678.19,E2 24678.19} C_VEL
LIN {X 0,Y 528.527,Z 274.386,A -85,B 0,C 180,E1 24674.834,E2 24674.834} C_VEL
LIN {X 0,Y 528.486,Z 274.403,A -85,B 0,C 180,E1 24671.458,E2 24671.458} C_VEL
LIN {X 0,Y 528.476,Z 274.394,A -85,B 0,C 180,E1 24668.048,E2 24668.048} C_VEL
LIN {X 0,Y 528.527,Z 274.395,A -85,B 0,C 180,E1 24664.775,E2 24664.775} C_VEL
LIN {X 0,Y 528.486,Z 274.394,A -85,B 0,C 180,E1 24661.409,E2 24661.409} C_VEL
LIN {X 0,Y 528.482,Z 274.395,A -85,B 0,C 180,E1 24657.94,E2 24657.94} C_VEL
LIN {X 0,Y 528.527,Z 274.4,A -85,B 0,C 180,E1 24654.572,E2 24654.572} C_VEL
LIN {X 0,Y 528.495,Z 274.395,A -85,B 0,C 180,E1 24651.185,E2 24651.185} C_VEL
LIN {X 0,Y 528.485,Z 274.4,A -85,B 0,C 180,E1 24647.767,E2 24647.767} C_VEL
LIN {X 0,Y 528.527,Z 274.387,A -85,B 0,C 180,E1 24644.417,E2 24644.417} C_VEL
LIN {X 0,Y 528.502,Z 274.404,A -85,B 0,C 180,E1 24641.01,E2 24641.01} C_VEL
LIN {X 0,Y 528.488,Z 274.401,A -85,B 0,C 180,E1 24637.532,E2 24637.532} C_VEL
LIN {X 0,Y 528.526,Z 274.398,A -85,B 0,C 180,E1 24634.208,E2 24634.208} C_VEL
LIN {X 0,Y 528.513,Z 274.403,A -85,B 0,C 180,E1 24630.785,E2 24630.785} C_VEL
LIN {X 0,Y 528.492,Z 274.401,A -85,B 0,C 180,E1 24627.339,E2 24627.339} C_VEL
LIN {X 0,Y 528.521,Z 274.398,A -85,B 0,C 180,E1 24623.879,E2 24623.879} C_VEL
LIN {X 0,Y 528.508,Z 274.398,A -85,B 0,C 180,E1 24621.622,E2 24621.622} C_VEL
LIN {X 0,Y 527.491,Z 274.531,A -85,B 0,C 180,E1 24620.787,E2 24620.787} C_VEL
LIN {X 0,Y 521.029,Z 275.335,A -85,B 0,C 180,E1 24618.38,E2 24618.38} C_VEL
LIN {X 0,Y 520.584,Z 275.387,A -85,B 0,C 180,E1 24617.829,E2 24617.829} C_VEL
LIN {X 0,Y 520.587,Z 275.39,A -85,B 0,C 180,E1 24614.354,E2 24614.354} C_VEL
LIN {X 0,Y 520.561,Z 275.391,A -85,B 0,C 180,E1 24610.916,E2 24610.916} C_VEL
LIN {X 0,Y 520.578,Z 275.386,A -85,B 0,C 180,E1 24607.505,E2 24607.505} C_VEL
LIN {X 0,Y 520.582,Z 275.391,A -85,B 0,C 180,E1 24604.112,E2 24604.112} C_VEL
LIN {X 0,Y 520.574,Z 275.39,A -85,B 0,C 180,E1 24600.595,E2 24600.595} C_VEL
LIN {X 0,Y 520.567,Z 275.386,A -85,B 0,C 180,E1 24597.078,E2 24597.078} C_VEL
LIN {X 0,Y 520.583,Z 275.386,A -85,B 0,C 180,E1 24593.631,E2 24593.631} C_VEL
LIN {X 0,Y 520.585,Z 275.39,A -85,B 0,C 180,E1 24590.084,E2 24590.084} C_VEL
LIN {X 0,Y 520.571,Z 275.391,A -85,B 0,C 180,E1 24586.58,E2 24586.58} C_VEL
LIN {X 0,Y 520.582,Z 275.386,A -85,B 0,C 180,E1 24583.099,E2 24583.099} C_VEL
LIN {X 0,Y 520.576,Z 275.39,A -85,B 0,C 180,E1 24579.619,E2 24579.619} C_VEL
LIN {X 0,Y 520.583,Z 275.39,A -85,B 0,C 180,E1 24576.174,E2 24576.174} C_VEL
LIN {X 0,Y 520.573,Z 275.388,A -85,B 0,C 180,E1 24572.642,E2 24572.642} C_VEL
LIN {X 0,Y 520.577,Z 275.385,A -85,B 0,C 180,E1 24569.23,E2 24569.23} C_VEL
LIN {X 0,Y 520.575,Z 275.39,A -85,B 0,C 180,E1 24565.704,E2 24565.704} C_VEL
LIN {X 0,Y 520.575,Z 275.391,A -85,B 0,C 180,E1 24562.274,E2 24562.274} C_VEL
LIN {X 0,Y 520.582,Z 275.386,A -85,B 0,C 180,E1 24558.815,E2 24558.815} C_VEL
LIN {X 0,Y 520.567,Z 275.39,A -85,B 0,C 180,E1 24555.314,E2 24555.314} C_VEL
LIN {X 0,Y 520.583,Z 275.39,A -85,B 0,C 180,E1 24551.872,E2 24551.872} C_VEL
LIN {X 0,Y 520.58,Z 275.387,A -85,B 0,C 180,E1 24548.361,E2 24548.361} C_VEL
LIN {X 0,Y 520.571,Z 275.386,A -85,B 0,C 180,E1 24544.883,E2 24544.883} C_VEL
LIN {X 0,Y 520.57,Z 275.39,A -85,B 0,C 180,E1 24541.373,E2 24541.373} C_VEL
LIN {X 0,Y 520.583,Z 275.389,A -85,B 0,C 180,E1 24537.989,E2 24537.989} C_VEL
LIN {X 0,Y 520.579,Z 275.386,A -85,B 0,C 180,E1 24534.524,E2 24534.524} C_VEL
LIN {X 0,Y 520.561,Z 275.391,A -85,B 0,C 180,E1 24531.068,E2 24531.068} C_VEL
LIN {X 0,Y 520.584,Z 275.391,A -85,B 0,C 180,E1 24527.614,E2 24527.614} C_VEL
LIN {X 0,Y 520.587,Z 275.387,A -85,B 0,C 180,E1 24524.086,E2 24524.086} C_VEL
LIN {X 0,Y 520.561,Z 275.389,A -85,B 0,C 180,E1 24520.627,E2 24520.627} C_VEL
LIN {X 0,Y 520.563,Z 275.393,A -85,B 0,C 180,E1 24517.093,E2 24517.093} C_VEL
LIN {X 0,Y 520.586,Z 275.39,A -85,B 0,C 180,E1 24513.715,E2 24513.715} C_VEL
LIN {X 0,Y 520.562,Z 275.388,A -85,B 0,C 180,E1 24510.341,E2 24510.341} C_VEL
LIN {X 0,Y 520.554,Z 275.391,A -85,B 0,C 180,E1 24506.832,E2 24506.832} C_VEL
LIN {X 0,Y 520.587,Z 275.392,A -85,B 0,C 180,E1 24503.359,E2 24503.359} C_VEL
LIN {X 0,Y 520.581,Z 275.386,A -85,B 0,C 180,E1 24499.874,E2 24499.874} C_VEL
LIN {X 0,Y 520.544,Z 275.381,A -85,B 0,C 180,E1 24496.516,E2 24496.516} C_VEL
LIN {X 0,Y 520.578,Z 275.392,A -85,B 0,C 180,E1 24493.099,E2 24493.099} C_VEL
LIN {X 0,Y 520.582,Z 275.373,A -85,B 0,C 180,E1 24489.619,E2 24489.619} C_VEL
LIN {X 0,Y 520.542,Z 275.39,A -85,B 0,C 180,E1 24486.286,E2 24486.286} C_VEL
LIN {X 0,Y 520.561,Z 275.379,A -85,B 0,C 180,E1 24482.862,E2 24482.862} C_VEL
LIN {X 0,Y 520.591,Z 275.387,A -85,B 0,C 180,E1 24479.45,E2 24479.45} C_VEL
LIN {X 0,Y 520.539,Z 275.383,A -85,B 0,C 180,E1 24476.035,E2 24476.035} C_VEL
LIN {X 0,Y 520.543,Z 275.384,A -85,B 0,C 180,E1 24472.495,E2 24472.495} C_VEL
LIN {X 0,Y 520.588,Z 275.383,A -85,B 0,C 180,E1 24469.151,E2 24469.151} C_VEL
LIN {X 0,Y 520.539,Z 275.382,A -85,B 0,C 180,E1 24465.767,E2 24465.767} C_VEL
LIN {X 0,Y 520.537,Z 275.393,A -85,B 0,C 180,E1 24462.307,E2 24462.307} C_VEL
LIN {X 0,Y 520.587,Z 275.375,A -85,B 0,C 180,E1 24458.952,E2 24458.952} C_VEL
LIN {X 0,Y 520.536,Z 275.389,A -85,B 0,C 180,E1 24455.608,E2 24455.608} C_VEL
LIN {X 0,Y 520.527,Z 275.394,A -85,B 0,C 180,E1 24452.076,E2 24452.076} C_VEL
LIN {X 0,Y 520.583,Z 275.386,A -85,B 0,C 180,E1 24448.763,E2 24448.763} C_VEL
LIN {X 0,Y 520.53,Z 275.389,A -85,B 0,C 180,E1 24445.483,E2 24445.483} C_VEL
LIN {X 0,Y 520.52,Z 275.366,A -85,B 0,C 180,E1 24441.956,E2 24441.956} C_VEL
LIN {X 0,Y 520.583,Z 275.393,A -85,B 0,C 180,E1 24438.647,E2 24438.647} C_VEL
LIN {X 0,Y 520.526,Z 275.371,A -85,B 0,C 180,E1 24435.292,E2 24435.292} C_VEL
LIN {X 0,Y 520.606,Z 275.621,A -85,B 0,C 180,E1 24432.499,E2 24432.499} C_VEL
LIN {X 0,Y 527.326,Z 295.432,A -85,B 0,C 180,E1 24429.292,E2 24429.292} C_VEL
LIN {X 0,Y 528.84,Z 301.019,A -85,B 0,C 180,E1 24428.463,E2 24428.463} C_VEL
LIN {X 0,Y 528.759,Z 305.75,A -85,B 0,C 180,E1 24427.929,E2 24427.929} C_VEL
LIN {X 0,Y 535.119,Z 327.843,A -85,B 0,C 180,E1 24427.037,E2 24427.037} C_VEL
LIN {X 0,Y 532.564,Z 545.144,A -85,B 0,C 180,E1 24423.719,E2 24423.719} C_VEL
LIN {X 0,Y 531.771,Z 608.31,A -85,B 0,C 180,E1 24422.737,E2 24422.737} C_VEL
LIN {X 0,Y 531.04,Z 631.469,A -85,B 0,C 180,E1 24422.177,E2 24422.177} C_VEL
LIN {X 0,Y 530.25,Z 651.711,A -85,B 0,C 180,E1 24421.487,E2 24421.487} C_VEL
LIN {X 0,Y 529.274,Z 672.201,A -85,B 0,C 180,E1 24420.604,E2 24420.604} C_VEL
LIN {X 0,Y 528.15,Z 691.727,A -85,B 0,C 180,E1 24419.548,E2 24419.548} C_VEL
LIN {X 0,Y 527.126,Z 709.177,A -85,B 0,C 180,E1 24418.43,E2 24418.43} C_VEL
LIN {X 0,Y 525.906,Z 728.389,A -85,B 0,C 180,E1 24416.985,E2 24416.985} C_VEL
LIN {X 0,Y 524.709,Z 746.261,A -85,B 0,C 180,E1 24415.387,E2 24415.387} C_VEL
LIN {X 0,Y 523.642,Z 763.186,A -85,B 0,C 180,E1 24413.639,E2 24413.639} C_VEL
LIN {X 0,Y 522.672,Z 778.521,A -85,B 0,C 180,E1 24411.784,E2 24411.784} C_VEL
LIN {X 0,Y 521.865,Z 792.553,A -85,B 0,C 180,E1 24409.827,E2 24409.827} C_VEL
LIN {X 0,Y 521.173,Z 805.914,A -85,B 0,C 180,E1 24407.645,E2 24407.645} C_VEL
LIN {X 0,Y 520.709,Z 816.641,A -85,B 0,C 180,E1 24405.594,E2 24405.594} C_VEL
LIN {X 0,Y 520.332,Z 827.1,A -85,B 0,C 180,E1 24403.218,E2 24403.218} C_VEL
LIN {X 0,Y 520.107,Z 835.112,A -85,B 0,C 180,E1 24400.971,E2 24400.971} C_VEL
LIN {X 0,Y 519.981,Z 841.873,A -85,B 0,C 180,E1 24398.626,E2 24398.626} C_VEL
LIN {X 0,Y 519.929,Z 846.834,A -85,B 0,C 180,E1 24396.293,E2 24396.293} C_VEL
LIN {X 0,Y 519.908,Z 850.366,A -85,B 0,C 180,E1 24393.859,E2 24393.859} C_VEL
LIN {X 0,Y 519.904,Z 852.215,A -85,B 0,C 180,E1 24391.322,E2 24391.322} C_VEL
LIN {X 0,Y 519.907,Z 852.322,A -85,B 0,C 180,E1 24389.118,E2 24389.118} C_VEL
LIN {X 0,Y 519.915,Z 850.927,A -85,B 0,C 180,E1 24386.693,E2 24386.693} C_VEL
LIN {X 0,Y 519.926,Z 847.784,A -85,B 0,C 180,E1 24384.261,E2 24384.261} C_VEL
LIN {X 0,Y 519.974,Z 843.334,A -85,B 0,C 180,E1 24382.009,E2 24382.009} C_VEL
LIN {X 0,Y 520.087,Z 836.541,A -85,B 0,C 180,E1 24379.477,E2 24379.477} C_VEL
LIN {X 0,Y 520.277,Z 828.807,A -85,B 0,C 180,E1 24377.232,E2 24377.232} C_VEL
LIN {X 0,Y 520.598,Z 819.331,A -85,B 0,C 180,E1 24374.973,E2 24374.973} C_VEL
LIN {X 0,Y 521.081,Z 807.811,A -85,B 0,C 180,E1 24372.698,E2 24372.698} C_VEL
LIN {X 0,Y 521.707,Z 795.595,A -85,B 0,C 180,E1 24370.637,E2 24370.637} C_VEL
LIN {X 0,Y 522.52,Z 781.176,A -85,B 0,C 180,E1 24368.563,E2 24368.563} C_VEL
LIN {X 0,Y 523.473,Z 765.717,A -85,B 0,C 180,E1 24366.651,E2 24366.651} C_VEL
LIN {X 0,Y 524.629,Z 747.484,A -85,B 0,C 180,E1 24364.729,E2 24364.729} C_VEL
LIN {X 0,Y 525.748,Z 730.681,A -85,B 0,C 180,E1 24363.211,E2 24363.211} C_VEL
LIN {X 0,Y 527.032,Z 710.731,A -85,B 0,C 180,E1 24361.675,E2 24361.675} C_VEL
LIN {X 0,Y 528.095,Z 692.709,A -85,B 0,C 180,E1 24360.511,E2 24360.511} C_VEL
LIN {X 0,Y 529.2,Z 673.361,A -85,B 0,C 180,E1 24359.454,E2 24359.454} C_VEL
LIN {X 0,Y 530.221,Z 652.492,A -85,B 0,C 180,E1 24358.543,E2 24358.543} C_VEL
LIN {X 0,Y 530.995,Z 632.543,A -85,B 0,C 180,E1 24357.856,E2 24357.856} C_VEL
LIN {X 0,Y 531.749,Z 609.768,A -85,B 0,C 180,E1 24357.289,E2 24357.289} C_VEL
LIN {X 0,Y 532.368,Z 562.527,A -85,B 0,C 180,E1 24356.543,E2 24356.543} C_VEL
LIN {X 0,Y 534.866,Z 348.002,A -85,B 0,C 180,E1 24353.274,E2 24353.274} C_VEL
LIN {X 0,Y 534.932,Z 326.647,A -85,B 0,C 180,E1 24352.928,E2 24352.928} C_VEL
LIN {X 0,Y 528.68,Z 305.075,A -85,B 0,C 180,E1 24352.023,E2 24352.023} C_VEL
LIN {X 0,Y 528.672,Z 299.724,A -85,B 0,C 180,E1 24351.36,E2 24351.36} C_VEL
LIN {X 0,Y 522.136,Z 280.484,A -85,B 0,C 180,E1 24348.316,E2 24348.316} C_VEL
LIN {X 0,Y 520.592,Z 275.515,A -85,B 0,C 180,E1 24347.465,E2 24347.465} C_VEL
LIN {X 0,Y 520.519,Z 275.366,A -85,B 0,C 180,E1 24344.078,E2 24344.078} C_VEL
LIN {X 0,Y 520.529,Z 275.392,A -85,B 0,C 180,E1 24340.63,E2 24340.63} C_VEL
LIN {X 0,Y 520.576,Z 275.368,A -85,B 0,C 180,E1 24337.332,E2 24337.332} C_VEL
LIN {X 0,Y 520.525,Z 275.39,A -85,B 0,C 180,E1 24333.985,E2 24333.985} C_VEL
LIN {X 0,Y 520.533,Z 275.383,A -85,B 0,C 180,E1 24330.471,E2 24330.471} C_VEL
LIN {X 0,Y 520.583,Z 275.385,A -85,B 0,C 180,E1 24327.201,E2 24327.201} C_VEL
LIN {X 0,Y 520.529,Z 275.39,A -85,B 0,C 180,E1 24323.894,E2 24323.894} C_VEL
LIN {X 0,Y 520.546,Z 275.377,A -85,B 0,C 180,E1 24320.462,E2 24320.462} C_VEL
LIN {X 0,Y 520.582,Z 275.387,A -85,B 0,C 180,E1 24317.089,E2 24317.089} C_VEL
LIN {X 0,Y 520.532,Z 275.382,A -85,B 0,C 180,E1 24313.779,E2 24313.779} C_VEL
LIN {X 0,Y 520.557,Z 275.381,A -85,B 0,C 180,E1 24310.402,E2 24310.402} C_VEL
LIN {X 0,Y 520.58,Z 275.386,A -85,B 0,C 180,E1 24307.061,E2 24307.061} C_VEL
LIN {X 0,Y 520.539,Z 275.384,A -85,B 0,C 180,E1 24303.634,E2 24303.634} C_VEL
LIN {X 0,Y 520.557,Z 275.389,A -85,B 0,C 180,E1 24300.22,E2 24300.22} C_VEL
LIN {X 0,Y 520.582,Z 275.374,A -85,B 0,C 180,E1 24296.807,E2 24296.807} C_VEL
LIN {X 0,Y 520.546,Z 275.392,A -85,B 0,C 180,E1 24293.382,E2 24293.382} C_VEL
LIN {X 0,Y 520.547,Z 275.377,A -85,B 0,C 180,E1 24289.822,E2 24289.822} C_VEL
LIN {X 0,Y 520.589,Z 275.383,A -85,B 0,C 180,E1 24286.449,E2 24286.449} C_VEL
LIN {X 0,Y 520.563,Z 275.383,A -85,B 0,C 180,E1 24283.025,E2 24283.025} C_VEL
LIN {X 0,Y 520.55,Z 275.389,A -85,B 0,C 180,E1 24279.538,E2 24279.538} C_VEL
LIN {X 0,Y 520.584,Z 275.387,A -85,B 0,C 180,E1 24276.093,E2 24276.093} C_VEL
LIN {X 0,Y 520.581,Z 275.393,A -85,B 0,C 180,E1 24272.675,E2 24272.675} C_VEL
LIN {X 0,Y 520.552,Z 275.391,A -85,B 0,C 180,E1 24269.275,E2 24269.275} C_VEL
LIN {X 0,Y 520.58,Z 275.387,A -85,B 0,C 180,E1 24265.872,E2 24265.872} C_VEL
LIN {X 0,Y 520.586,Z 275.39,A -85,B 0,C 180,E1 24262.355,E2 24262.355} C_VEL
LIN {X 0,Y 520.561,Z 275.392,A -85,B 0,C 180,E1 24258.937,E2 24258.937} C_VEL
LIN {X 0,Y 520.584,Z 275.387,A -85,B 0,C 180,E1 24257.829,E2 24257.829} C_VEL
LIN {X 0,Y 519.577,Z 275.514,A -85,B 0,C 180,E1 24256.982,E2 24256.982} C_VEL
LIN {X 0,Y 513.169,Z 276.316,A -85,B 0,C 180,E1 24254.6,E2 24254.6} C_VEL
LIN {X 0,Y 512.647,Z 276.377,A -85,B 0,C 180,E1 24253.979,E2 24253.979} C_VEL
LIN {X 0,Y 512.645,Z 276.379,A -85,B 0,C 180,E1 24250.478,E2 24250.478} C_VEL
LIN {X 0,Y 512.623,Z 276.378,A -85,B 0,C 180,E1 24247.062,E2 24247.062} C_VEL
LIN {X 0,Y 512.645,Z 276.375,A -85,B 0,C 180,E1 24243.611,E2 24243.611} C_VEL
LIN {X 0,Y 512.646,Z 276.379,A -85,B 0,C 180,E1 24240.082,E2 24240.082} C_VEL
LIN {X 0,Y 512.63,Z 276.378,A -85,B 0,C 180,E1 24236.653,E2 24236.653} C_VEL
LIN {X 0,Y 512.633,Z 276.375,A -85,B 0,C 180,E1 24233.081,E2 24233.081} C_VEL
LIN {X 0,Y 512.642,Z 276.377,A -85,B 0,C 180,E1 24229.6,E2 24229.6} C_VEL
LIN {X 0,Y 512.645,Z 276.379,A -85,B 0,C 180,E1 24226.078,E2 24226.078} C_VEL
LIN {X 0,Y 512.631,Z 276.38,A -85,B 0,C 180,E1 24222.618,E2 24222.618} C_VEL
LIN {X 0,Y 512.645,Z 276.375,A -85,B 0,C 180,E1 24219.09,E2 24219.09} C_VEL
LIN {X 0,Y 512.635,Z 276.379,A -85,B 0,C 180,E1 24215.596,E2 24215.596} C_VEL
LIN {X 0,Y 512.643,Z 276.38,A -85,B 0,C 180,E1 24212.124,E2 24212.124} C_VEL
LIN {X 0,Y 512.637,Z 276.375,A -85,B 0,C 180,E1 24208.659,E2 24208.659} C_VEL
LIN {X 0,Y 512.638,Z 276.376,A -85,B 0,C 180,E1 24205.189,E2 24205.189} C_VEL
LIN {X 0,Y 512.64,Z 276.379,A -85,B 0,C 180,E1 24201.702,E2 24201.702} C_VEL
LIN {X 0,Y 512.641,Z 276.38,A -85,B 0,C 180,E1 24198.183,E2 24198.183} C_VEL
LIN {X 0,Y 512.647,Z 276.376,A -85,B 0,C 180,E1 24194.619,E2 24194.619} C_VEL
LIN {X 0,Y 512.631,Z 276.377,A -85,B 0,C 180,E1 24191.078,E2 24191.078} C_VEL
LIN {X 0,Y 512.635,Z 276.381,A -85,B 0,C 180,E1 24187.525,E2 24187.525} C_VEL
LIN {X 0,Y 512.643,Z 276.377,A -85,B 0,C 180,E1 24184.044,E2 24184.044} C_VEL
LIN {X 0,Y 512.645,Z 276.373,A -85,B 0,C 180,E1 24180.562,E2 24180.562} C_VEL
LIN {X 0,Y 512.625,Z 276.378,A -85,B 0,C 180,E1 24177.032,E2 24177.032} C_VEL
LIN {X 0,Y 512.64,Z 276.379,A -85,B 0,C 180,E1 24173.472,E2 24173.472} C_VEL
LIN {X 0,Y 512.645,Z 276.378,A -85,B 0,C 180,E1 24170.041,E2 24170.041} C_VEL
LIN {X 0,Y 512.626,Z 276.377,A -85,B 0,C 180,E1 24166.643,E2 24166.643} C_VEL
LIN {X 0,Y 512.625,Z 276.382,A -85,B 0,C 180,E1 24163.159,E2 24163.159} C_VEL
LIN {X 0,Y 512.647,Z 276.38,A -85,B 0,C 180,E1 24159.771,E2 24159.771} C_VEL
LIN {X 0,Y 512.63,Z 276.377,A -85,B 0,C 180,E1 24156.34,E2 24156.34} C_VEL
LIN {X 0,Y 512.616,Z 276.38,A -85,B 0,C 180,E1 24152.836,E2 24152.836} C_VEL
LIN {X 0,Y 512.648,Z 276.379,A -85,B 0,C 180,E1 24149.439,E2 24149.439} C_VEL
LIN {X 0,Y 512.645,Z 276.376,A -85,B 0,C 180,E1 24145.905,E2 24145.905} C_VEL
LIN {X 0,Y 512.611,Z 276.379,A -85,B 0,C 180,E1 24142.476,E2 24142.476} C_VEL
LIN {X 0,Y 512.626,Z 276.382,A -85,B 0,C 180,E1 24139.01,E2 24139.01} C_VEL
LIN {X 0,Y 512.649,Z 276.361,A -85,B 0,C 180,E1 24135.537,E2 24135.537} C_VEL
LIN {X 0,Y 512.611,Z 276.378,A -85,B 0,C 180,E1 24132.161,E2 24132.161} C_VEL
LIN {X 0,Y 512.608,Z 276.373,A -85,B 0,C 180,E1 24128.638,E2 24128.638} C_VEL
LIN {X 0,Y 512.647,Z 276.374,A -85,B 0,C 180,E1 24125.26,E2 24125.26} C_VEL
LIN {X 0,Y 512.621,Z 276.371,A -85,B 0,C 180,E1 24121.788,E2 24121.788} C_VEL
LIN {X 0,Y 512.602,Z 276.37,A -85,B 0,C 180,E1 24118.435,E2 24118.435} C_VEL
LIN {X 0,Y 512.645,Z 276.375,A -85,B 0,C 180,E1 24115.077,E2 24115.077} C_VEL
LIN {X 0,Y 512.613,Z 276.369,A -85,B 0,C 180,E1 24111.701,E2 24111.701} C_VEL
LIN {X 0,Y 512.597,Z 276.381,A -85,B 0,C 180,E1 24108.282,E2 24108.282} C_VEL
LIN {X 0,Y 512.637,Z 276.364,A -85,B 0,C 180,E1 24104.849,E2 24104.849} C_VEL
LIN {X 0,Y 512.621,Z 276.379,A -85,B 0,C 180,E1 24101.425,E2 24101.425} C_VEL
LIN {X 0,Y 512.589,Z 276.379,A -85,B 0,C 180,E1 24098.006,E2 24098.006} C_VEL
LIN {X 0,Y 512.621,Z 276.367,A -85,B 0,C 180,E1 24094.589,E2 24094.589} C_VEL
LIN {X 0,Y 512.625,Z 276.381,A -85,B 0,C 180,E1 24091.199,E2 24091.199} C_VEL
LIN {X 0,Y 512.585,Z 276.383,A -85,B 0,C 180,E1 24087.824,E2 24087.824} C_VEL
LIN {X 0,Y 512.615,Z 276.382,A -85,B 0,C 180,E1 24084.423,E2 24084.423} C_VEL
LIN {X 0,Y 512.612,Z 276.346,A -85,B 0,C 180,E1 24081.093,E2 24081.093} C_VEL
LIN {X 0,Y 512.579,Z 276.38,A -85,B 0,C 180,E1 24077.836,E2 24077.836} C_VEL
LIN {X 0,Y 512.625,Z 276.372,A -85,B 0,C 180,E1 24074.443,E2 24074.443} C_VEL
LIN {X 0,Y 512.643,Z 276.673,A -85,B 0,C 180,E1 24073.112,E2 24073.112} C_VEL
LIN {X 0,Y 518.508,Z 294.057,A -85,B 0,C 180,E1 24070.216,E2 24070.216} C_VEL
LIN {X 0,Y 521.608,Z 303.933,A -85,B 0,C 180,E1 24068.674,E2 24068.674} C_VEL
LIN {X 0,Y 521.831,Z 306.004,A -85,B 0,C 180,E1 24068.514,E2 24068.514} C_VEL
LIN {X 0,Y 528.694,Z 329.934,A -85,B 0,C 180,E1 24067.526,E2 24067.526} C_VEL
LIN {X 0,Y 525.897,Z 546.431,A -85,B 0,C 180,E1 24064.184,E2 24064.184} C_VEL
LIN {X 0,Y 525.038,Z 608.289,A -85,B 0,C 180,E1 24063.211,E2 24063.211} C_VEL
LIN {X 0,Y 524.245,Z 631.446,A -85,B 0,C 180,E1 24062.645,E2 24062.645} C_VEL
LIN {X 0,Y 523.413,Z 650.681,A -85,B 0,C 180,E1 24061.988,E2 24061.988} C_VEL
LIN {X 0,Y 522.379,Z 670.938,A -85,B 0,C 180,E1 24061.116,E2 24061.116} C_VEL
LIN {X 0,Y 521.071,Z 691.721,A -85,B 0,C 180,E1 24059.99,E2 24059.99} C_VEL
LIN {X 0,Y 519.946,Z 709.168,A -85,B 0,C 180,E1 24058.859,E2 24058.859} C_VEL
LIN {X 0,Y 518.574,Z 728.623,A -85,B 0,C 180,E1 24057.377,E2 24057.377} C_VEL
LIN {X 0,Y 517.353,Z 745.38,A -85,B 0,C 180,E1 24055.863,E2 24055.863} C_VEL
LIN {X 0,Y 516.19,Z 761.712,A -85,B 0,C 180,E1 24054.172,E2 24054.172} C_VEL
LIN {X 0,Y 515.034,Z 778.119,A -85,B 0,C 180,E1 24052.178,E2 24052.178} C_VEL
LIN {X 0,Y 514.155,Z 791.809,A -85,B 0,C 180,E1 24050.251,E2 24050.251} C_VEL
LIN {X 0,Y 513.343,Z 805.913,A -85,B 0,C 180,E1 24047.923,E2 24047.923} C_VEL
LIN {X 0,Y 512.819,Z 816.636,A -85,B 0,C 180,E1 24045.84,E2 24045.84} C_VEL
LIN {X 0,Y 512.393,Z 827.099,A -85,B 0,C 180,E1 24043.427,E2 24043.427} C_VEL
LIN {X 0,Y 512.137,Z 835.109,A -85,B 0,C 180,E1 24041.144,E2 24041.144} C_VEL
LIN {X 0,Y 511.992,Z 841.872,A -85,B 0,C 180,E1 24038.761,E2 24038.761} C_VEL
LIN {X 0,Y 511.93,Z 846.83,A -85,B 0,C 180,E1 24036.392,E2 24036.392} C_VEL
LIN {X 0,Y 511.909,Z 850.367,A -85,B 0,C 180,E1 24033.92,E2 24033.92} C_VEL
LIN {X 0,Y 511.903,Z 852.213,A -85,B 0,C 180,E1 24031.343,E2 24031.343} C_VEL
LIN {X 0,Y 511.908,Z 852.32,A -85,B 0,C 180,E1 24029.105,E2 24029.105} C_VEL
LIN {X 0,Y 511.915,Z 850.93,A -85,B 0,C 180,E1 24026.641,E2 24026.641} C_VEL
LIN {X 0,Y 511.927,Z 847.78,A -85,B 0,C 180,E1 24024.171,E2 24024.171} C_VEL
LIN {X 0,Y 511.982,Z 843.41,A -85,B 0,C 180,E1 24021.917,E2 24021.917} C_VEL
LIN {X 0,Y 512.103,Z 836.896,A -85,B 0,C 180,E1 24019.425,E2 24019.425} C_VEL
LIN {X 0,Y 512.312,Z 829.228,A -85,B 0,C 180,E1 24017.145,E2 24017.145} C_VEL
LIN {X 0,Y 512.667,Z 819.854,A -85,B 0,C 180,E1 24014.851,E2 24014.851} C_VEL
LIN {X 0,Y 513.201,Z 808.439,A -85,B 0,C 180,E1 24012.541,E2 24012.541} C_VEL
LIN {X 0,Y 513.841,Z 797.011,A -85,B 0,C 180,E1 24010.565,E2 24010.565} C_VEL
LIN {X 0,Y 514.79,Z 782.054,A -85,B 0,C 180,E1 24008.345,E2 24008.345} C_VEL
LIN {X 0,Y 515.831,Z 766.698,A -85,B 0,C 180,E1 24006.406,E2 24006.406} C_VEL
LIN {X 0,Y 517.108,Z 748.7,A -85,B 0,C 180,E1 24004.458,E2 24004.458} C_VEL
LIN {X 0,Y 518.296,Z 732.39,A -85,B 0,C 180,E1 24002.95,E2 24002.95} C_VEL
LIN {X 0,Y 519.665,Z 713.427,A -85,B 0,C 180,E1 24001.438,E2 24001.438} C_VEL
LIN {X 0,Y 520.946,Z 693.753,A -85,B 0,C 180,E1 24000.134,E2 24000.134} C_VEL
LIN {X 0,Y 522.07,Z 675.611,A -85,B 0,C 180,E1 23999.119,E2 23999.119} C_VEL
LIN {X 0,Y 523.31,Z 653.253,A -85,B 0,C 180,E1 23998.111,E2 23998.111} C_VEL
LIN {X 0,Y 524.142,Z 633.712,A -85,B 0,C 180,E1 23997.425,E2 23997.425} C_VEL
LIN {X 0,Y 524.969,Z 611.935,A -85,B 0,C 180,E1 23996.857,E2 23996.857} C_VEL
LIN {X 0,Y 525.551,Z 574.91,A -85,B 0,C 180,E1 23996.25,E2 23996.25} C_VEL
LIN {X 0,Y 528.303,Z 358.888,A -85,B 0,C 180,E1 23992.925,E2 23992.925} C_VEL
LIN {X 0,Y 528.509,Z 328.625,A -85,B 0,C 180,E1 23992.437,E2 23992.437} C_VEL
LIN {X 0,Y 521.598,Z 304.713,A -85,B 0,C 180,E1 23991.413,E2 23991.413} C_VEL
LIN {X 0,Y 521.213,Z 302.096,A -85,B 0,C 180,E1 23991.058,E2 23991.058} C_VEL
LIN {X 0,Y 515.177,Z 284.26,A -85,B 0,C 180,E1 23988.182,E2 23988.182} C_VEL
LIN {X 0,Y 512.609,Z 276.486,A -85,B 0,C 180,E1 23986.822,E2 23986.822} C_VEL
LIN {X 0,Y 512.626,Z 276.348,A -85,B 0,C 180,E1 23983.485,E2 23983.485} C_VEL
LIN {X 0,Y 512.58,Z 276.374,A -85,B 0,C 180,E1 23980.215,E2 23980.215} C_VEL
LIN {X 0,Y 512.617,Z 276.368,A -85,B 0,C 180,E1 23976.9,E2 23976.9} C_VEL
LIN {X 0,Y 512.61,Z 276.375,A -85,B 0,C 180,E1 23973.607,E2 23973.607} C_VEL
LIN {X 0,Y 512.586,Z 276.372,A -85,B 0,C 180,E1 23970.216,E2 23970.216} C_VEL
LIN {X 0,Y 512.637,Z 276.369,A -85,B 0,C 180,E1 23966.904,E2 23966.904} C_VEL
LIN {X 0,Y 512.608,Z 276.38,A -85,B 0,C 180,E1 23963.548,E2 23963.548} C_VEL
LIN {X 0,Y 512.59,Z 276.366,A -85,B 0,C 180,E1 23960.078,E2 23960.078} C_VEL
LIN {X 0,Y 512.632,Z 276.371,A -85,B 0,C 180,E1 23956.661,E2 23956.661} C_VEL
LIN {X 0,Y 512.624,Z 276.372,A -85,B 0,C 180,E1 23953.28,E2 23953.28} C_VEL
LIN {X 0,Y 512.595,Z 276.371,A -85,B 0,C 180,E1 23949.884,E2 23949.884} C_VEL
LIN {X 0,Y 512.633,Z 276.378,A -85,B 0,C 180,E1 23946.495,E2 23946.495} C_VEL
LIN {X 0,Y 512.636,Z 276.362,A -85,B 0,C 180,E1 23943.019,E2 23943.019} C_VEL
LIN {X 0,Y 512.601,Z 276.38,A -85,B 0,C 180,E1 23939.665,E2 23939.665} C_VEL
LIN {X 0,Y 512.622,Z 276.365,A -85,B 0,C 180,E1 23936.198,E2 23936.198} C_VEL
LIN {X 0,Y 512.652,Z 276.375,A -85,B 0,C 180,E1 23932.717,E2 23932.717} C_VEL
LIN {X 0,Y 512.609,Z 276.368,A -85,B 0,C 180,E1 23929.321,E2 23929.321} C_VEL
LIN {X 0,Y 512.611,Z 276.372,A -85,B 0,C 180,E1 23925.773,E2 23925.773} C_VEL
LIN {X 0,Y 512.649,Z 276.378,A -85,B 0,C 180,E1 23922.404,E2 23922.404} C_VEL
LIN {X 0,Y 512.627,Z 276.381,A -85,B 0,C 180,E1 23918.968,E2 23918.968} C_VEL
LIN {X 0,Y 512.612,Z 276.379,A -85,B 0,C 180,E1 23915.452,E2 23915.452} C_VEL
LIN {X 0,Y 512.641,Z 276.376,A -85,B 0,C 180,E1 23911.963,E2 23911.963} C_VEL
LIN {X 0,Y 512.648,Z 276.379,A -85,B 0,C 180,E1 23908.462,E2 23908.462} C_VEL
LIN {X 0,Y 512.621,Z 276.381,A -85,B 0,C 180,E1 23905.003,E2 23905.003} C_VEL
LIN {X 0,Y 512.622,Z 276.378,A -85,B 0,C 180,E1 23901.455,E2 23901.455} C_VEL
LIN {X 0,Y 512.647,Z 276.377,A -85,B 0,C 180,E1 23897.994,E2 23897.994} C_VEL
LIN {X 0,Y 512.645,Z 276.379,A -85,B 0,C 180,E1 23894.441,E2 23894.441} C_VEL
LIN {X 0,Y 512.647,Z 276.377,A -85,B 0,C 180,E1 23893.979,E2 23893.979} C_VEL
LIN {X 0,Y 511.666,Z 276.499,A -85,B 0,C 180,E1 23893.119,E2 23893.119} C_VEL
LIN {X 0,Y 505.141,Z 277.319,A -85,B 0,C 180,E1 23890.637,E2 23890.637} C_VEL
LIN {X 0,Y 504.706,Z 277.368,A -85,B 0,C 180,E1 23890.069,E2 23890.069} C_VEL
LIN {X 0,Y 504.696,Z 277.368,A -85,B 0,C 180,E1 23886.605,E2 23886.605} C_VEL
LIN {X 0,Y 504.688,Z 277.367,A -85,B 0,C 180,E1 23883.011,E2 23883.011} C_VEL
LIN {X 0,Y 504.712,Z 277.362,A -85,B 0,C 180,E1 23879.556,E2 23879.556} C_VEL
LIN {X 0,Y 504.705,Z 277.366,A -85,B 0,C 180,E1 23875.964,E2 23875.964} C_VEL
LIN {X 0,Y 504.696,Z 277.37,A -85,B 0,C 180,E1 23872.479,E2 23872.479} C_VEL
LIN {X 0,Y 504.693,Z 277.366,A -85,B 0,C 180,E1 23868.959,E2 23868.959} C_VEL
LIN {X 0,Y 504.708,Z 277.365,A -85,B 0,C 180,E1 23865.394,E2 23865.394} C_VEL
LIN {X 0,Y 504.703,Z 277.369,A -85,B 0,C 180,E1 23861.86,E2 23861.86} C_VEL
LIN {X 0,Y 504.7,Z 277.368,A -85,B 0,C 180,E1 23858.315,E2 23858.315} C_VEL
LIN {X 0,Y 504.698,Z 277.366,A -85,B 0,C 180,E1 23854.773,E2 23854.773} C_VEL
LIN {X 0,Y 504.702,Z 277.363,A -85,B 0,C 180,E1 23851.249,E2 23851.249} C_VEL
LIN {X 0,Y 504.7,Z 277.367,A -85,B 0,C 180,E1 23847.729,E2 23847.729} C_VEL
LIN {X 0,Y 504.7,Z 277.37,A -85,B 0,C 180,E1 23844.201,E2 23844.201} C_VEL
LIN {X 0,Y 504.703,Z 277.366,A -85,B 0,C 180,E1 23840.601,E2 23840.601} C_VEL
LIN {X 0,Y 504.698,Z 277.366,A -85,B 0,C 180,E1 23837.064,E2 23837.064} C_VEL
LIN {X 0,Y 504.696,Z 277.37,A -85,B 0,C 180,E1 23833.507,E2 23833.507} C_VEL
LIN {X 0,Y 504.705,Z 277.367,A -85,B 0,C 180,E1 23829.958,E2 23829.958} C_VEL
LIN {X 0,Y 504.707,Z 277.364,A -85,B 0,C 180,E1 23826.412,E2 23826.412} C_VEL
LIN {X 0,Y 504.691,Z 277.364,A -85,B 0,C 180,E1 23822.893,E2 23822.893} C_VEL
LIN {X 0,Y 504.691,Z 277.367,A -85,B 0,C 180,E1 23819.295,E2 23819.295} C_VEL
LIN {X 0,Y 504.708,Z 277.37,A -85,B 0,C 180,E1 23815.764,E2 23815.764} C_VEL
LIN {X 0,Y 504.708,Z 277.365,A -85,B 0,C 180,E1 23812.227,E2 23812.227} C_VEL
LIN {X 0,Y 504.687,Z 277.367,A -85,B 0,C 180,E1 23808.723,E2 23808.723} C_VEL
LIN {X 0,Y 504.688,Z 277.37,A -85,B 0,C 180,E1 23805.149,E2 23805.149} C_VEL
LIN {X 0,Y 504.708,Z 277.368,A -85,B 0,C 180,E1 23801.683,E2 23801.683} C_VEL
LIN {X 0,Y 504.708,Z 277.365,A -85,B 0,C 180,E1 23798.144,E2 23798.144} C_VEL
LIN {X 0,Y 504.677,Z 277.368,A -85,B 0,C 180,E1 23794.652,E2 23794.652} C_VEL
LIN {X 0,Y 504.691,Z 277.371,A -85,B 0,C 180,E1 23791.136,E2 23791.136} C_VEL
LIN {X 0,Y 504.71,Z 277.368,A -85,B 0,C 180,E1 23787.617,E2 23787.617} C_VEL
LIN {X 0,Y 504.693,Z 277.366,A -85,B 0,C 180,E1 23784.086,E2 23784.086} C_VEL
LIN {X 0,Y 504.672,Z 277.368,A -85,B 0,C 180,E1 23780.65,E2 23780.65} C_VEL
LIN {X 0,Y 504.699,Z 277.361,A -85,B 0,C 180,E1 23777.168,E2 23777.168} C_VEL
LIN {X 0,Y 504.71,Z 277.359,A -85,B 0,C 180,E1 23773.636,E2 23773.636} C_VEL
LIN {X 0,Y 504.671,Z 277.353,A -85,B 0,C 180,E1 23770.156,E2 23770.156} C_VEL
LIN {X 0,Y 504.668,Z 277.37,A -85,B 0,C 180,E1 23766.598,E2 23766.598} C_VEL
LIN {X 0,Y 504.703,Z 277.348,A -85,B 0,C 180,E1 23763.18,E2 23763.18} C_VEL
LIN {X 0,Y 504.68,Z 277.367,A -85,B 0,C 180,E1 23759.773,E2 23759.773} C_VEL
LIN {X 0,Y 504.661,Z 277.36,A -85,B 0,C 180,E1 23756.365,E2 23756.365} C_VEL
LIN {X 0,Y 504.702,Z 277.362,A -85,B 0,C 180,E1 23752.945,E2 23752.945} C_VEL
LIN {X 0,Y 504.688,Z 277.358,A -85,B 0,C 180,E1 23749.498,E2 23749.498} C_VEL
LIN {X 0,Y 504.653,Z 277.36,A -85,B 0,C 180,E1 23746.12,E2 23746.12} C_VEL
LIN {X 0,Y 504.688,Z 277.372,A -85,B 0,C 180,E1 23742.712,E2 23742.712} C_VEL
LIN {X 0,Y 504.683,Z 277.351,A -85,B 0,C 180,E1 23739.351,E2 23739.351} C_VEL
LIN {X 0,Y 504.651,Z 277.368,A -85,B 0,C 180,E1 23735.972,E2 23735.972} C_VEL
LIN {X 0,Y 504.677,Z 277.371,A -85,B 0,C 180,E1 23732.509,E2 23732.509} C_VEL
LIN {X 0,Y 504.688,Z 277.359,A -85,B 0,C 180,E1 23729.129,E2 23729.129} C_VEL
LIN {X 0,Y 504.645,Z 277.367,A -85,B 0,C 180,E1 23725.709,E2 23725.709} C_VEL
LIN {X 0,Y 504.657,Z 277.34,A -85,B 0,C 180,E1 23722.232,E2 23722.232} C_VEL
LIN {X 0,Y 504.705,Z 277.369,A -85,B 0,C 180,E1 23718.832,E2 23718.832} C_VEL
LIN {X 0,Y 504.641,Z 277.342,A -85,B 0,C 180,E1 23715.462,E2 23715.462} C_VEL
LIN {X 0,Y 504.683,Z 277.667,A -85,B 0,C 180,E1 23713.763,E2 23713.763} C_VEL
LIN {X 0,Y 510.3,Z 294.011,A -85,B 0,C 180,E1 23710.946,E2 23710.946} C_VEL
LIN {X 0,Y 513.883,Z 304.663,A -85,B 0,C 180,E1 23709.251,E2 23709.251} C_VEL
LIN {X 0,Y 515.86,Z 309.232,A -85,B 0,C 180,E1 23708.981,E2 23708.981} C_VEL
LIN {X 0,Y 522.305,Z 331.977,A -85,B 0,C 180,E1 23708.027,E2 23708.027} C_VEL
LIN {X 0,Y 519.263,Z 547.933,A -85,B 0,C 180,E1 23704.658,E2 23704.658} C_VEL
LIN {X 0,Y 518.343,Z 608.268,A -85,B 0,C 180,E1 23703.697,E2 23703.697} C_VEL
LIN {X 0,Y 517.489,Z 631.422,A -85,B 0,C 180,E1 23703.126,E2 23703.126} C_VEL
LIN {X 0,Y 516.593,Z 650.268,A -85,B 0,C 180,E1 23702.479,E2 23702.479} C_VEL
LIN {X 0,Y 515.507,Z 669.953,A -85,B 0,C 180,E1 23701.629,E2 23701.629} C_VEL
LIN {X 0,Y 514.104,Z 690.732,A -85,B 0,C 180,E1 23700.504,E2 23700.504} C_VEL
LIN {X 0,Y 512.866,Z 708.123,A -85,B 0,C 180,E1 23699.373,E2 23699.373} C_VEL
LIN {X 0,Y 511.404,Z 727.364,A -85,B 0,C 180,E1 23697.906,E2 23697.906} C_VEL
LIN {X 0,Y 509.985,Z 745.027,A -85,B 0,C 180,E1 23696.3,E2 23696.3} C_VEL
LIN {X 0,Y 508.755,Z 760.502,A -85,B 0,C 180,E1 23694.684,E2 23694.684} C_VEL
LIN {X 0,Y 507.514,Z 776.738,A -85,B 0,C 180,E1 23692.714,E2 23692.714} C_VEL
LIN {X 0,Y 506.477,Z 791.016,A -85,B 0,C 180,E1 23690.693,E2 23690.693} C_VEL
LIN {X 0,Y 505.562,Z 805.299,A -85,B 0,C 180,E1 23688.323,E2 23688.323} C_VEL
LIN {X 0,Y 504.948,Z 816.189,A -85,B 0,C 180,E1 23686.187,E2 23686.187} C_VEL
LIN {X 0,Y 504.475,Z 826.646,A -85,B 0,C 180,E1 23683.759,E2 23683.759} C_VEL
LIN {X 0,Y 504.172,Z 835.105,A -85,B 0,C 180,E1 23681.322,E2 23681.322} C_VEL
LIN {X 0,Y 504.008,Z 841.872,A -85,B 0,C 180,E1 23678.901,E2 23678.901} C_VEL
LIN {X 0,Y 503.933,Z 846.826,A -85,B 0,C 180,E1 23676.494,E2 23676.494} C_VEL
LIN {X 0,Y 503.914,Z 850.229,A -85,B 0,C 180,E1 23674.096,E2 23674.096} C_VEL
LIN {X 0,Y 503.898,Z 852.157,A -85,B 0,C 180,E1 23671.592,E2 23671.592} C_VEL
LIN {X 0,Y 503.903,Z 852.345,A -85,B 0,C 180,E1 23669.204,E2 23669.204} C_VEL
LIN {X 0,Y 503.916,Z 851.129,A -85,B 0,C 180,E1 23666.815,E2 23666.815} C_VEL
LIN {X 0,Y 503.928,Z 847.966,A -85,B 0,C 180,E1 23664.192,E2 23664.192} C_VEL
LIN {X 0,Y 503.988,Z 843.593,A -85,B 0,C 180,E1 23661.874,E2 23661.874} C_VEL
LIN {X 0,Y 504.119,Z 837.252,A -85,B 0,C 180,E1 23659.371,E2 23659.371} C_VEL
LIN {X 0,Y 504.348,Z 829.65,A -85,B 0,C 180,E1 23657.055,E2 23657.055} C_VEL
LIN {X 0,Y 504.739,Z 820.377,A -85,B 0,C 180,E1 23654.725,E2 23654.725} C_VEL
LIN {X 0,Y 505.326,Z 809.067,A -85,B 0,C 180,E1 23652.379,E2 23652.379} C_VEL
LIN {X 0,Y 506.025,Z 797.719,A -85,B 0,C 180,E1 23650.373,E2 23650.373} C_VEL
LIN {X 0,Y 507.003,Z 783.773,A -85,B 0,C 180,E1 23648.239,E2 23648.239} C_VEL
LIN {X 0,Y 508.118,Z 768.662,A -85,B 0,C 180,E1 23646.272,E2 23646.272} C_VEL
LIN {X 0,Y 509.374,Z 752.815,A -85,B 0,C 180,E1 23644.479,E2 23644.479} C_VEL
LIN {X 0,Y 510.805,Z 734.763,A -85,B 0,C 180,E1 23642.74,E2 23642.74} C_VEL
LIN {X 0,Y 512.162,Z 717.341,A -85,B 0,C 180,E1 23641.299,E2 23641.299} C_VEL
LIN {X 0,Y 513.706,Z 696.624,A -85,B 0,C 180,E1 23639.858,E2 23639.858} C_VEL
LIN {X 0,Y 514.895,Z 678.988,A -85,B 0,C 180,E1 23638.836,E2 23638.836} C_VEL
LIN {X 0,Y 516.107,Z 659.726,A -85,B 0,C 180,E1 23637.904,E2 23637.904} C_VEL
LIN {X 0,Y 517.228,Z 637.345,A -85,B 0,C 180,E1 23637.061,E2 23637.061} C_VEL
LIN {X 0,Y 517.982,Z 618.253,A -85,B 0,C 180,E1 23636.521,E2 23636.521} C_VEL
LIN {X 0,Y 518.638,Z 595.646,A -85,B 0,C 180,E1 23636.078,E2 23636.078} C_VEL
LIN {X 0,Y 521.704,Z 373.301,A -85,B 0,C 180,E1 23632.624,E2 23632.624} C_VEL
LIN {X 0,Y 522.141,Z 330.74,A -85,B 0,C 180,E1 23631.938,E2 23631.938} C_VEL
LIN {X 0,Y 515.097,Z 307.146,A -85,B 0,C 180,E1 23630.914,E2 23630.914} C_VEL
LIN {X 0,Y 513.682,Z 304.133,A -85,B 0,C 180,E1 23630.689,E2 23630.689} C_VEL
LIN {X 0,Y 507.402,Z 285.569,A -85,B 0,C 180,E1 23627.631,E2 23627.631} C_VEL
LIN {X 0,Y 504.658,Z 277.495,A -85,B 0,C 180,E1 23626.181,E2 23626.181} C_VEL
LIN {X 0,Y 504.65,Z 277.351,A -85,B 0,C 180,E1 23622.69,E2 23622.69} C_VEL
LIN {X 0,Y 504.701,Z 277.333,A -85,B 0,C 180,E1 23619.342,E2 23619.342} C_VEL
LIN {X 0,Y 504.651,Z 277.371,A -85,B 0,C 180,E1 23615.906,E2 23615.906} C_VEL
LIN {X 0,Y 504.649,Z 277.372,A -85,B 0,C 180,E1 23612.34,E2 23612.34} C_VEL
LIN {X 0,Y 504.707,Z 277.366,A -85,B 0,C 180,E1 23609.036,E2 23609.036} C_VEL
LIN {X 0,Y 504.666,Z 277.355,A -85,B 0,C 180,E1 23605.589,E2 23605.589} C_VEL
LIN {X 0,Y 504.651,Z 277.367,A -85,B 0,C 180,E1 23602.114,E2 23602.114} C_VEL
LIN {X 0,Y 504.694,Z 277.366,A -85,B 0,C 180,E1 23598.72,E2 23598.72} C_VEL
LIN {X 0,Y 504.688,Z 277.351,A -85,B 0,C 180,E1 23595.25,E2 23595.25} C_VEL
LIN {X 0,Y 504.657,Z 277.369,A -85,B 0,C 180,E1 23591.842,E2 23591.842} C_VEL
LIN {X 0,Y 504.685,Z 277.354,A -85,B 0,C 180,E1 23588.43,E2 23588.43} C_VEL
LIN {X 0,Y 504.702,Z 277.365,A -85,B 0,C 180,E1 23585.001,E2 23585.001} C_VEL
LIN {X 0,Y 504.662,Z 277.358,A -85,B 0,C 180,E1 23581.589,E2 23581.589} C_VEL
LIN {X 0,Y 504.673,Z 277.36,A -85,B 0,C 180,E1 23578.07,E2 23578.07} C_VEL
LIN {X 0,Y 504.709,Z 277.364,A -85,B 0,C 180,E1 23574.657,E2 23574.657} C_VEL
LIN {X 0,Y 504.676,Z 277.358,A -85,B 0,C 180,E1 23571.225,E2 23571.225} C_VEL
LIN {X 0,Y 504.669,Z 277.367,A -85,B 0,C 180,E1 23567.761,E2 23567.761} C_VEL
LIN {X 0,Y 504.708,Z 277.349,A -85,B 0,C 180,E1 23564.317,E2 23564.317} C_VEL
LIN {X 0,Y 504.701,Z 277.37,A -85,B 0,C 180,E1 23560.8,E2 23560.8} C_VEL
LIN {X 0,Y 504.673,Z 277.369,A -85,B 0,C 180,E1 23557.397,E2 23557.397} C_VEL
LIN {X 0,Y 504.696,Z 277.365,A -85,B 0,C 180,E1 23553.909,E2 23553.909} C_VEL
LIN {X 0,Y 504.71,Z 277.367,A -85,B 0,C 180,E1 23550.419,E2 23550.419} C_VEL
LIN {X 0,Y 504.687,Z 277.371,A -85,B 0,C 180,E1 23546.93,E2 23546.93} C_VEL
LIN {X 0,Y 504.68,Z 277.368,A -85,B 0,C 180,E1 23543.355,E2 23543.355} C_VEL
LIN {X 0,Y 504.707,Z 277.365,A -85,B 0,C 180,E1 23539.878,E2 23539.878} C_VEL
LIN {X 0,Y 504.708,Z 277.368,A -85,B 0,C 180,E1 23536.308,E2 23536.308} C_VEL
LIN {X 0,Y 504.688,Z 277.37,A -85,B 0,C 180,E1 23532.806,E2 23532.806} C_VEL
LIN {X 0,Y 504.706,Z 277.368,A -85,B 0,C 180,E1 23530.069,E2 23530.069} C_VEL
LIN {X 0,Y 503.721,Z 277.488,A -85,B 0,C 180,E1 23529.194,E2 23529.194} C_VEL
LIN {X 0,Y 497.204,Z 278.309,A -85,B 0,C 180,E1 23526.673,E2 23526.673} C_VEL
LIN {X 0,Y 496.766,Z 278.358,A -85,B 0,C 180,E1 23526.096,E2 23526.096} C_VEL
LIN {X 0,Y 496.76,Z 278.357,A -85,B 0,C 180,E1 23522.505,E2 23522.505} C_VEL
LIN {X 0,Y 496.75,Z 278.354,A -85,B 0,C 180,E1 23519.017,E2 23519.017} C_VEL
LIN {X 0,Y 496.766,Z 278.352,A -85,B 0,C 180,E1 23515.513,E2 23515.513} C_VEL
LIN {X 0,Y 496.764,Z 278.355,A -85,B 0,C 180,E1 23511.895,E2 23511.895} C_VEL
LIN {X 0,Y 496.764,Z 278.358,A -85,B 0,C 180,E1 23508.299,E2 23508.299} C_VEL
LIN {X 0,Y 496.754,Z 278.357,A -85,B 0,C 180,E1 23504.81,E2 23504.81} C_VEL
LIN {X 0,Y 496.766,Z 278.354,A -85,B 0,C 180,E1 23501.258,E2 23501.258} C_VEL
LIN {X 0,Y 496.76,Z 278.359,A -85,B 0,C 180,E1 23497.75,E2 23497.75} C_VEL
LIN {X 0,Y 496.76,Z 278.356,A -85,B 0,C 180,E1 23494.271,E2 23494.271} C_VEL
LIN {X 0,Y 496.758,Z 278.353,A -85,B 0,C 180,E1 23490.692,E2 23490.692} C_VEL
LIN {X 0,Y 496.763,Z 278.353,A -85,B 0,C 180,E1 23487.116,E2 23487.116} C_VEL
LIN {X 0,Y 496.756,Z 278.356,A -85,B 0,C 180,E1 23483.528,E2 23483.528} C_VEL
LIN {X 0,Y 496.765,Z 278.357,A -85,B 0,C 180,E1 23480.032,E2 23480.032} C_VEL
LIN {X 0,Y 496.763,Z 278.356,A -85,B 0,C 180,E1 23476.447,E2 23476.447} C_VEL
LIN {X 0,Y 496.76,Z 278.355,A -85,B 0,C 180,E1 23472.911,E2 23472.911} C_VEL
LIN {X 0,Y 496.752,Z 278.358,A -85,B 0,C 180,E1 23469.376,E2 23469.376} C_VEL
LIN {X 0,Y 496.768,Z 278.357,A -85,B 0,C 180,E1 23465.885,E2 23465.885} C_VEL
LIN {X 0,Y 496.766,Z 278.352,A -85,B 0,C 180,E1 23462.294,E2 23462.294} C_VEL
LIN {X 0,Y 496.753,Z 278.354,A -85,B 0,C 180,E1 23458.807,E2 23458.807} C_VEL
LIN {X 0,Y 496.75,Z 278.357,A -85,B 0,C 180,E1 23455.207,E2 23455.207} C_VEL
LIN {X 0,Y 496.772,Z 278.357,A -85,B 0,C 180,E1 23451.691,E2 23451.691} C_VEL
LIN {X 0,Y 496.769,Z 278.356,A -85,B 0,C 180,E1 23448.071,E2 23448.071} C_VEL
LIN {X 0,Y 496.751,Z 278.355,A -85,B 0,C 180,E1 23444.561,E2 23444.561} C_VEL
LIN {X 0,Y 496.743,Z 278.359,A -85,B 0,C 180,E1 23440.993,E2 23440.993} C_VEL
LIN {X 0,Y 496.768,Z 278.356,A -85,B 0,C 180,E1 23437.534,E2 23437.534} C_VEL
LIN {X 0,Y 496.768,Z 278.355,A -85,B 0,C 180,E1 23433.981,E2 23433.981} C_VEL
LIN {X 0,Y 496.742,Z 278.356,A -85,B 0,C 180,E1 23430.48,E2 23430.48} C_VEL
LIN {X 0,Y 496.741,Z 278.359,A -85,B 0,C 180,E1 23426.917,E2 23426.917} C_VEL
LIN {X 0,Y 496.771,Z 278.359,A -85,B 0,C 180,E1 23423.36,E2 23423.36} C_VEL
LIN {X 0,Y 496.769,Z 278.354,A -85,B 0,C 180,E1 23419.763,E2 23419.763} C_VEL
LIN {X 0,Y 496.733,Z 278.344,A -85,B 0,C 180,E1 23416.237,E2 23416.237} C_VEL
LIN {X 0,Y 496.732,Z 278.359,A -85,B 0,C 180,E1 23412.674,E2 23412.674} C_VEL
LIN {X 0,Y 496.763,Z 278.337,A -85,B 0,C 180,E1 23409.149,E2 23409.149} C_VEL
LIN {X 0,Y 496.762,Z 278.355,A -85,B 0,C 180,E1 23405.66,E2 23405.66} C_VEL
LIN {X 0,Y 496.725,Z 278.35,A -85,B 0,C 180,E1 23402.192,E2 23402.192} C_VEL
LIN {X 0,Y 496.732,Z 278.347,A -85,B 0,C 180,E1 23398.616,E2 23398.616} C_VEL
LIN {X 0,Y 496.77,Z 278.35,A -85,B 0,C 180,E1 23395.151,E2 23395.151} C_VEL
LIN {X 0,Y 496.729,Z 278.346,A -85,B 0,C 180,E1 23391.783,E2 23391.783} C_VEL
LIN {X 0,Y 496.72,Z 278.359,A -85,B 0,C 180,E1 23388.27,E2 23388.27} C_VEL
LIN {X 0,Y 496.756,Z 278.339,A -85,B 0,C 180,E1 23384.831,E2 23384.831} C_VEL
LIN {X 0,Y 496.751,Z 278.357,A -85,B 0,C 180,E1 23381.335,E2 23381.335} C_VEL
LIN {X 0,Y 496.713,Z 278.357,A -85,B 0,C 180,E1 23377.888,E2 23377.888} C_VEL
LIN {X 0,Y 496.724,Z 278.343,A -85,B 0,C 180,E1 23374.356,E2 23374.356} C_VEL
LIN {X 0,Y 496.773,Z 278.351,A -85,B 0,C 180,E1 23370.852,E2 23370.852} C_VEL
LIN {X 0,Y 496.726,Z 278.36,A -85,B 0,C 180,E1 23367.353,E2 23367.353} C_VEL
LIN {X 0,Y 496.706,Z 278.359,A -85,B 0,C 180,E1 23363.857,E2 23363.857} C_VEL
LIN {X 0,Y 496.736,Z 278.326,A -85,B 0,C 180,E1 23360.435,E2 23360.435} C_VEL
LIN {X 0,Y 496.725,Z 278.331,A -85,B 0,C 180,E1 23357.111,E2 23357.111} C_VEL
LIN {X 0,Y 496.778,Z 278.571,A -85,B 0,C 180,E1 23354.459,E2 23354.459} C_VEL
LIN {X 0,Y 502.071,Z 294.136,A -85,B 0,C 180,E1 23351.686,E2 23351.686} C_VEL
LIN {X 0,Y 505.45,Z 304.122,A -85,B 0,C 180,E1 23350.045,E2 23350.045} C_VEL
LIN {X 0,Y 509.929,Z 312.451,A -85,B 0,C 180,E1 23349.461,E2 23349.461} C_VEL
LIN {X 0,Y 515.956,Z 334.024,A -85,B 0,C 180,E1 23348.541,E2 23348.541} C_VEL
LIN {X 0,Y 512.65,Z 549.605,A -85,B 0,C 180,E1 23345.14,E2 23345.14} C_VEL
LIN {X 0,Y 511.68,Z 608.302,A -85,B 0,C 180,E1 23344.194,E2 23344.194} C_VEL
LIN {X 0,Y 510.771,Z 631.399,A -85,B 0,C 180,E1 23343.619,E2 23343.619} C_VEL
LIN {X 0,Y 509.807,Z 650.093,A -85,B 0,C 180,E1 23342.972,E2 23342.972} C_VEL
LIN {X 0,Y 508.671,Z 668.978,A -85,B 0,C 180,E1 23342.153,E2 23342.153} C_VEL
LIN {X 0,Y 507.11,Z 690.725,A -85,B 0,C 180,E1 23340.97,E2 23340.97} C_VEL
LIN {X 0,Y 505.804,Z 707.42,A -85,B 0,C 180,E1 23339.876,E2 23339.876} C_VEL
LIN {X 0,Y 504.316,Z 725.758,A -85,B 0,C 180,E1 23338.477,E2 23338.477} C_VEL
LIN {X 0,Y 502.715,Z 743.799,A -85,B 0,C 180,E1 23336.838,E2 23336.838} C_VEL
LIN {X 0,Y 501.412,Z 758.853,A -85,B 0,C 180,E1 23335.26,E2 23335.26} C_VEL
LIN {X 0,Y 500.068,Z 774.947,A -85,B 0,C 180,E1 23333.321,E2 23333.321} C_VEL
LIN {X 0,Y 498.874,Z 789.505,A -85,B 0,C 180,E1 23331.257,E2 23331.257} C_VEL
LIN {X 0,Y 497.932,Z 802.676,A -85,B 0,C 180,E1 23329.105,E2 23329.105} C_VEL
LIN {X 0,Y 497.163,Z 814.523,A -85,B 0,C 180,E1 23326.805,E2 23326.805} C_VEL
LIN {X 0,Y 496.618,Z 824.862,A -85,B 0,C 180,E1 23324.44,E2 23324.44} C_VEL
LIN {X 0,Y 496.241,Z 834.011,A -85,B 0,C 180,E1 23321.859,E2 23321.859} C_VEL
LIN {X 0,Y 496.061,Z 840.103,A -85,B 0,C 180,E1 23319.727,E2 23319.727} C_VEL
LIN {X 0,Y 495.965,Z 845.608,A -85,B 0,C 180,E1 23317.296,E2 23317.296} C_VEL
LIN {X 0,Y 495.921,Z 849.55,A -85,B 0,C 180,E1 23314.742,E2 23314.742} C_VEL
LIN {X 0,Y 495.909,Z 851.77,A -85,B 0,C 180,E1 23312.311,E2 23312.311} C_VEL
LIN {X 0,Y 495.9,Z 852.44,A -85,B 0,C 180,E1 23309.653,E2 23309.653} C_VEL
LIN {X 0,Y 495.909,Z 851.529,A -85,B 0,C 180,E1 23307.342,E2 23307.342} C_VEL
LIN {X 0,Y 495.926,Z 849.063,A -85,B 0,C 180,E1 23304.856,E2 23304.856} C_VEL
LIN {X 0,Y 495.976,Z 844.637,A -85,B 0,C 180,E1 23302.238,E2 23302.238} C_VEL
LIN {X 0,Y 496.076,Z 839.442,A -85,B 0,C 180,E1 23300.018,E2 23300.018} C_VEL
LIN {X 0,Y 496.315,Z 832.141,A -85,B 0,C 180,E1 23297.552,E2 23297.552} C_VEL
LIN {X 0,Y 496.694,Z 823.322,A -85,B 0,C 180,E1 23295.188,E2 23295.188} C_VEL
LIN {X 0,Y 497.247,Z 813.273,A -85,B 0,C 180,E1 23292.928,E2 23292.928} C_VEL
LIN {X 0,Y 498.065,Z 800.554,A -85,B 0,C 180,E1 23290.535,E2 23290.535} C_VEL
LIN {X 0,Y 498.94,Z 788.631,A -85,B 0,C 180,E1 23288.61,E2 23288.61} C_VEL
LIN {X 0,Y 500.141,Z 774.019,A -85,B 0,C 180,E1 23286.558,E2 23286.558} C_VEL
LIN {X 0,Y 501.459,Z 758.304,A -85,B 0,C 180,E1 23284.68,E2 23284.68} C_VEL
LIN {X 0,Y 502.77,Z 743.187,A -85,B 0,C 180,E1 23283.101,E2 23283.101} C_VEL
LIN {X 0,Y 504.423,Z 724.391,A -85,B 0,C 180,E1 23281.414,E2 23281.414} C_VEL
LIN {X 0,Y 505.872,Z 706.556,A -85,B 0,C 180,E1 23280.063,E2 23280.063} C_VEL
LIN {X 0,Y 507.372,Z 687.778,A -85,B 0,C 180,E1 23278.85,E2 23278.85} C_VEL
LIN {X 0,Y 508.779,Z 667.006,A -85,B 0,C 180,E1 23277.755,E2 23277.755} C_VEL
LIN {X 0,Y 509.851,Z 649.312,A -85,B 0,C 180,E1 23276.998,E2 23276.998} C_VEL
LIN {X 0,Y 510.892,Z 629.36,A -85,B 0,C 180,E1 23276.318,E2 23276.318} C_VEL
LIN {X 0,Y 511.712,Z 606.633,A -85,B 0,C 180,E1 23275.775,E2 23275.775} C_VEL
LIN {X 0,Y 514.223,Z 445.155,A -85,B 0,C 180,E1 23273.223,E2 23273.223} C_VEL
LIN {X 0,Y 515.786,Z 332.691,A -85,B 0,C 180,E1 23271.421,E2 23271.421} C_VEL
LIN {X 0,Y 509.354,Z 311.142,A -85,B 0,C 180,E1 23270.463,E2 23270.463} C_VEL
LIN {X 0,Y 505.287,Z 303.753,A -85,B 0,C 180,E1 23269.911,E2 23269.911} C_VEL
LIN {X 0,Y 499.698,Z 286.989,A -85,B 0,C 180,E1 23267.083,E2 23267.083} C_VEL
LIN {X 0,Y 496.769,Z 278.482,A -85,B 0,C 180,E1 23265.504,E2 23265.504} C_VEL
LIN {X 0,Y 496.704,Z 278.355,A -85,B 0,C 180,E1 23262.092,E2 23262.092} C_VEL
LIN {X 0,Y 496.711,Z 278.32,A -85,B 0,C 180,E1 23258.61,E2 23258.61} C_VEL
LIN {X 0,Y 496.766,Z 278.356,A -85,B 0,C 180,E1 23255.145,E2 23255.145} C_VEL
LIN {X 0,Y 496.73,Z 278.362,A -85,B 0,C 180,E1 23251.633,E2 23251.633} C_VEL
LIN {X 0,Y 496.711,Z 278.361,A -85,B 0,C 180,E1 23248.158,E2 23248.158} C_VEL
LIN {X 0,Y 496.748,Z 278.349,A -85,B 0,C 180,E1 23244.75,E2 23244.75} C_VEL
LIN {X 0,Y 496.744,Z 278.344,A -85,B 0,C 180,E1 23241.366,E2 23241.366} C_VEL
LIN {X 0,Y 496.715,Z 278.357,A -85,B 0,C 180,E1 23237.937,E2 23237.937} C_VEL
LIN {X 0,Y 496.738,Z 278.341,A -85,B 0,C 180,E1 23234.453,E2 23234.453} C_VEL
LIN {X 0,Y 496.764,Z 278.351,A -85,B 0,C 180,E1 23231.023,E2 23231.023} C_VEL
LIN {X 0,Y 496.727,Z 278.349,A -85,B 0,C 180,E1 23227.518,E2 23227.518} C_VEL
LIN {X 0,Y 496.722,Z 278.349,A -85,B 0,C 180,E1 23223.924,E2 23223.924} C_VEL
LIN {X 0,Y 496.763,Z 278.355,A -85,B 0,C 180,E1 23220.461,E2 23220.461} C_VEL
LIN {X 0,Y 496.754,Z 278.338,A -85,B 0,C 180,E1 23217,E2 23217} C_VEL
LIN {X 0,Y 496.727,Z 278.358,A -85,B 0,C 180,E1 23213.528,E2 23213.528} C_VEL
LIN {X 0,Y 496.742,Z 278.339,A -85,B 0,C 180,E1 23210.032,E2 23210.032} C_VEL
LIN {X 0,Y 496.773,Z 278.35,A -85,B 0,C 180,E1 23206.498,E2 23206.498} C_VEL
LIN {X 0,Y 496.752,Z 278.348,A -85,B 0,C 180,E1 23202.95,E2 23202.95} C_VEL
LIN {X 0,Y 496.733,Z 278.357,A -85,B 0,C 180,E1 23199.498,E2 23199.498} C_VEL
LIN {X 0,Y 496.761,Z 278.354,A -85,B 0,C 180,E1 23196.01,E2 23196.01} C_VEL
LIN {X 0,Y 496.771,Z 278.357,A -85,B 0,C 180,E1 23192.424,E2 23192.424} C_VEL
LIN {X 0,Y 496.745,Z 278.36,A -85,B 0,C 180,E1 23188.984,E2 23188.984} C_VEL
LIN {X 0,Y 496.74,Z 278.357,A -85,B 0,C 180,E1 23185.409,E2 23185.409} C_VEL
LIN {X 0,Y 496.769,Z 278.354,A -85,B 0,C 180,E1 23181.837,E2 23181.837} C_VEL
LIN {X 0,Y 496.769,Z 278.357,A -85,B 0,C 180,E1 23178.225,E2 23178.225} C_VEL
LIN {X 0,Y 496.76,Z 278.357,A -85,B 0,C 180,E1 23174.623,E2 23174.623} C_VEL
LIN {X 0,Y 496.745,Z 278.357,A -85,B 0,C 180,E1 23171.161,E2 23171.161} C_VEL
LIN {X 0,Y 496.769,Z 278.354,A -85,B 0,C 180,E1 23167.721,E2 23167.721} C_VEL
LIN {X 0,Y 496.766,Z 278.358,A -85,B 0,C 180,E1 23166.096,E2 23166.096} C_VEL
LIN {X 0,Y 495.779,Z 278.476,A -85,B 0,C 180,E1 23165.207,E2 23165.207} C_VEL
LIN {X 0,Y 489.266,Z 279.297,A -85,B 0,C 180,E1 23162.645,E2 23162.645} C_VEL
LIN {X 0,Y 488.828,Z 279.346,A -85,B 0,C 180,E1 23162.058,E2 23162.058} C_VEL
LIN {X 0,Y 488.823,Z 279.346,A -85,B 0,C 180,E1 23158.462,E2 23158.462} C_VEL
LIN {X 0,Y 488.812,Z 279.343,A -85,B 0,C 180,E1 23154.92,E2 23154.92} C_VEL
LIN {X 0,Y 488.83,Z 279.342,A -85,B 0,C 180,E1 23151.351,E2 23151.351} C_VEL
LIN {X 0,Y 488.825,Z 279.344,A -85,B 0,C 180,E1 23147.744,E2 23147.744} C_VEL
LIN {X 0,Y 488.834,Z 279.344,A -85,B 0,C 180,E1 23144.087,E2 23144.087} C_VEL
LIN {X 0,Y 488.817,Z 279.346,A -85,B 0,C 180,E1 23140.489,E2 23140.489} C_VEL
LIN {X 0,Y 488.827,Z 279.343,A -85,B 0,C 180,E1 23136.931,E2 23136.931} C_VEL
LIN {X 0,Y 488.82,Z 279.344,A -85,B 0,C 180,E1 23133.401,E2 23133.401} C_VEL
LIN {X 0,Y 488.824,Z 279.345,A -85,B 0,C 180,E1 23129.766,E2 23129.766} C_VEL
LIN {X 0,Y 488.824,Z 279.348,A -85,B 0,C 180,E1 23126.13,E2 23126.13} C_VEL
LIN {X 0,Y 488.823,Z 279.344,A -85,B 0,C 180,E1 23122.596,E2 23122.596} C_VEL
LIN {X 0,Y 488.821,Z 279.344,A -85,B 0,C 180,E1 23119.034,E2 23119.034} C_VEL
LIN {X 0,Y 488.814,Z 279.348,A -85,B 0,C 180,E1 23115.429,E2 23115.429} C_VEL
LIN {X 0,Y 488.828,Z 279.345,A -85,B 0,C 180,E1 23111.887,E2 23111.887} C_VEL
LIN {X 0,Y 488.826,Z 279.343,A -85,B 0,C 180,E1 23108.221,E2 23108.221} C_VEL
LIN {X 0,Y 488.824,Z 279.341,A -85,B 0,C 180,E1 23104.692,E2 23104.692} C_VEL
LIN {X 0,Y 488.81,Z 279.344,A -85,B 0,C 180,E1 23101.101,E2 23101.101} C_VEL
LIN {X 0,Y 488.825,Z 279.346,A -85,B 0,C 180,E1 23097.596,E2 23097.596} C_VEL
LIN {X 0,Y 488.828,Z 279.345,A -85,B 0,C 180,E1 23094.054,E2 23094.054} C_VEL
LIN {X 0,Y 488.825,Z 279.343,A -85,B 0,C 180,E1 23090.455,E2 23090.455} C_VEL
LIN {X 0,Y 488.805,Z 279.347,A -85,B 0,C 180,E1 23086.907,E2 23086.907} C_VEL
LIN {X 0,Y 488.823,Z 279.345,A -85,B 0,C 180,E1 23083.414,E2 23083.414} C_VEL
LIN {X 0,Y 488.831,Z 279.346,A -85,B 0,C 180,E1 23079.808,E2 23079.808} C_VEL
LIN {X 0,Y 488.82,Z 279.344,A -85,B 0,C 180,E1 23076.238,E2 23076.238} C_VEL
LIN {X 0,Y 488.799,Z 279.347,A -85,B 0,C 180,E1 23072.685,E2 23072.685} C_VEL
LIN {X 0,Y 488.815,Z 279.347,A -85,B 0,C 180,E1 23069.132,E2 23069.132} C_VEL
LIN {X 0,Y 488.832,Z 279.347,A -85,B 0,C 180,E1 23065.568,E2 23065.568} C_VEL
LIN {X 0,Y 488.822,Z 279.344,A -85,B 0,C 180,E1 23061.982,E2 23061.982} C_VEL
LIN {X 0,Y 488.794,Z 279.347,A -85,B 0,C 180,E1 23058.485,E2 23058.485} C_VEL
LIN {X 0,Y 488.804,Z 279.33,A -85,B 0,C 180,E1 23054.936,E2 23054.936} C_VEL
LIN {X 0,Y 488.833,Z 279.34,A -85,B 0,C 180,E1 23051.444,E2 23051.444} C_VEL
LIN {X 0,Y 488.807,Z 279.338,A -85,B 0,C 180,E1 23047.877,E2 23047.877} C_VEL
LIN {X 0,Y 488.786,Z 279.332,A -85,B 0,C 180,E1 23044.341,E2 23044.341} C_VEL
LIN {X 0,Y 488.805,Z 279.349,A -85,B 0,C 180,E1 23040.82,E2 23040.82} C_VEL
LIN {X 0,Y 488.829,Z 279.322,A -85,B 0,C 180,E1 23037.304,E2 23037.304} C_VEL
LIN {X 0,Y 488.795,Z 279.346,A -85,B 0,C 180,E1 23033.776,E2 23033.776} C_VEL
LIN {X 0,Y 488.779,Z 279.335,A -85,B 0,C 180,E1 23030.225,E2 23030.225} C_VEL
LIN {X 0,Y 488.809,Z 279.338,A -85,B 0,C 180,E1 23026.756,E2 23026.756} C_VEL
LIN {X 0,Y 488.824,Z 279.338,A -85,B 0,C 180,E1 23023.237,E2 23023.237} C_VEL
LIN {X 0,Y 488.777,Z 279.331,A -85,B 0,C 180,E1 23019.775,E2 23019.775} C_VEL
LIN {X 0,Y 488.78,Z 279.347,A -85,B 0,C 180,E1 23016.235,E2 23016.235} C_VEL
LIN {X 0,Y 488.82,Z 279.34,A -85,B 0,C 180,E1 23012.73,E2 23012.73} C_VEL
LIN {X 0,Y 488.788,Z 279.337,A -85,B 0,C 180,E1 23009.38,E2 23009.38} C_VEL
LIN {X 0,Y 488.768,Z 279.343,A -85,B 0,C 180,E1 23005.909,E2 23005.909} C_VEL
LIN {X 0,Y 488.797,Z 279.313,A -85,B 0,C 180,E1 23002.441,E2 23002.441} C_VEL
LIN {X 0,Y 488.804,Z 279.347,A -85,B 0,C 180,E1 22999.006,E2 22999.006} C_VEL
LIN {X 0,Y 488.76,Z 279.313,A -85,B 0,C 180,E1 22995.556,E2 22995.556} C_VEL
LIN {X 0,Y 488.852,Z 279.768,A -85,B 0,C 180,E1 22995.119,E2 22995.119} C_VEL
LIN {X 0,Y 494.41,Z 295.874,A -85,B 0,C 180,E1 22992.175,E2 22992.175} C_VEL
LIN {X 0,Y 497.067,Z 303.788,A -85,B 0,C 180,E1 22990.859,E2 22990.859} C_VEL
LIN {X 0,Y 504.256,Z 316.501,A -85,B 0,C 180,E1 22989.916,E2 22989.916} C_VEL
LIN {X 0,Y 509.652,Z 335.944,A -85,B 0,C 180,E1 22989.069,E2 22989.069} C_VEL
LIN {X 0,Y 506.073,Z 551.072,A -85,B 0,C 180,E1 22985.636,E2 22985.636} C_VEL
LIN {X 0,Y 505.044,Z 608.156,A -85,B 0,C 180,E1 22984.705,E2 22984.705} C_VEL
LIN {X 0,Y 504.069,Z 631.281,A -85,B 0,C 180,E1 22984.122,E2 22984.122} C_VEL
LIN {X 0,Y 503.037,Z 649.922,A -85,B 0,C 180,E1 22983.474,E2 22983.474} C_VEL
LIN {X 0,Y 501.815,Z 668.896,A -85,B 0,C 180,E1 22982.646,E2 22982.646} C_VEL
LIN {X 0,Y 500.247,Z 689.736,A -85,B 0,C 180,E1 22981.51,E2 22981.51} C_VEL
LIN {X 0,Y 498.808,Z 706.547,A -85,B 0,C 180,E1 22980.406,E2 22980.406} C_VEL
LIN {X 0,Y 497.309,Z 723.451,A -85,B 0,C 180,E1 22979.113,E2 22979.113} C_VEL
LIN {X 0,Y 495.507,Z 742.571,A -85,B 0,C 180,E1 22977.391,E2 22977.391} C_VEL
LIN {X 0,Y 494.048,Z 757.989,A -85,B 0,C 180,E1 22975.764,E2 22975.764} C_VEL
LIN {X 0,Y 492.574,Z 774.023,A -85,B 0,C 180,E1 22973.824,E2 22973.824} C_VEL
LIN {X 0,Y 491.263,Z 788.626,A -85,B 0,C 180,E1 22971.741,E2 22971.741} C_VEL
LIN {X 0,Y 490.302,Z 800.552,A -85,B 0,C 180,E1 22969.786,E2 22969.786} C_VEL
LIN {X 0,Y 489.396,Z 813.268,A -85,B 0,C 180,E1 22967.354,E2 22967.354} C_VEL
LIN {X 0,Y 488.782,Z 823.317,A -85,B 0,C 180,E1 22965.057,E2 22965.057} C_VEL
LIN {X 0,Y 488.348,Z 832.547,A -85,B 0,C 180,E1 22962.534,E2 22962.534} C_VEL
LIN {X 0,Y 488.099,Z 839.441,A -85,B 0,C 180,E1 22960.146,E2 22960.146} C_VEL
LIN {X 0,Y 487.988,Z 844.634,A -85,B 0,C 180,E1 22957.89,E2 22957.89} C_VEL
LIN {X 0,Y 487.927,Z 848.983,A -85,B 0,C 180,E1 22955.291,E2 22955.291} C_VEL
LIN {X 0,Y 487.91,Z 851.444,A -85,B 0,C 180,E1 22952.819,E2 22952.819} C_VEL
LIN {X 0,Y 487.898,Z 852.417,A -85,B 0,C 180,E1 22950.47,E2 22950.47} C_VEL
LIN {X 0,Y 487.91,Z 851.843,A -85,B 0,C 180,E1 22947.769,E2 22947.769} C_VEL
LIN {X 0,Y 487.92,Z 849.816,A -85,B 0,C 180,E1 22945.416,E2 22945.416} C_VEL
LIN {X 0,Y 487.967,Z 846.227,A -85,B 0,C 180,E1 22942.938,E2 22942.938} C_VEL
LIN {X 0,Y 488.068,Z 840.657,A -85,B 0,C 180,E1 22940.33,E2 22940.33} C_VEL
LIN {X 0,Y 488.254,Z 834.735,A -85,B 0,C 180,E1 22938.184,E2 22938.184} C_VEL
LIN {X 0,Y 488.633,Z 826.191,A -85,B 0,C 180,E1 22935.665,E2 22935.665} C_VEL
LIN {X 0,Y 489.203,Z 816.063,A -85,B 0,C 180,E1 22933.251,E2 22933.251} C_VEL
LIN {X 0,Y 489.952,Z 805.27,A -85,B 0,C 180,E1 22931.067,E2 22931.067} C_VEL
LIN {X 0,Y 491.068,Z 791.006,A -85,B 0,C 180,E1 22928.626,E2 22928.626} C_VEL
LIN {X 0,Y 492.24,Z 777.61,A -85,B 0,C 180,E1 22926.667,E2 22926.667} C_VEL
LIN {X 0,Y 493.771,Z 761.043,A -85,B 0,C 180,E1 22924.578,E2 22924.578} C_VEL
LIN {X 0,Y 495.204,Z 745.711,A -85,B 0,C 180,E1 22922.925,E2 22922.925} C_VEL
LIN {X 0,Y 496.77,Z 729.28,A -85,B 0,C 180,E1 22921.379,E2 22921.379} C_VEL
LIN {X 0,Y 498.555,Z 709.587,A -85,B 0,C 180,E1 22919.811,E2 22919.811} C_VEL
LIN {X 0,Y 499.978,Z 692.682,A -85,B 0,C 180,E1 22918.672,E2 22918.672} C_VEL
LIN {X 0,Y 501.435,Z 674.424,A -85,B 0,C 180,E1 22917.631,E2 22917.631} C_VEL
LIN {X 0,Y 502.902,Z 652.288,A -85,B 0,C 180,E1 22916.619,E2 22916.619} C_VEL
LIN {X 0,Y 503.923,Z 633.793,A -85,B 0,C 180,E1 22915.956,E2 22915.956} C_VEL
LIN {X 0,Y 504.901,Z 613.074,A -85,B 0,C 180,E1 22915.396,E2 22915.396} C_VEL
LIN {X 0,Y 505.604,Z 581.418,A -85,B 0,C 180,E1 22914.843,E2 22914.843} C_VEL
LIN {X 0,Y 509.18,Z 363.109,A -85,B 0,C 180,E1 22911.369,E2 22911.369} C_VEL
LIN {X 0,Y 509.502,Z 334.798,A -85,B 0,C 180,E1 22910.897,E2 22910.897} C_VEL
LIN {X 0,Y 503.647,Z 315.092,A -85,B 0,C 180,E1 22910.001,E2 22910.001} C_VEL
LIN {X 0,Y 496.853,Z 303.253,A -85,B 0,C 180,E1 22909.082,E2 22909.082} C_VEL
LIN {X 0,Y 491.637,Z 287.793,A -85,B 0,C 180,E1 22906.386,E2 22906.386} C_VEL
LIN {X 0,Y 488.794,Z 279.453,A -85,B 0,C 180,E1 22904.782,E2 22904.782} C_VEL
LIN {X 0,Y 488.828,Z 279.348,A -85,B 0,C 180,E1 22901.351,E2 22901.351} C_VEL
LIN {X 0,Y 488.774,Z 279.311,A -85,B 0,C 180,E1 22897.852,E2 22897.852} C_VEL
LIN {X 0,Y 488.77,Z 279.345,A -85,B 0,C 180,E1 22894.375,E2 22894.375} C_VEL
LIN {X 0,Y 488.812,Z 279.336,A -85,B 0,C 180,E1 22890.892,E2 22890.892} C_VEL
LIN {X 0,Y 488.796,Z 279.348,A -85,B 0,C 180,E1 22887.535,E2 22887.535} C_VEL
LIN {X 0,Y 488.774,Z 279.345,A -85,B 0,C 180,E1 22884.022,E2 22884.022} C_VEL
LIN {X 0,Y 488.8,Z 279.325,A -85,B 0,C 180,E1 22880.599,E2 22880.599} C_VEL
LIN {X 0,Y 488.822,Z 279.342,A -85,B 0,C 180,E1 22877.13,E2 22877.13} C_VEL
LIN {X 0,Y 488.78,Z 279.336,A -85,B 0,C 180,E1 22873.678,E2 22873.678} C_VEL
LIN {X 0,Y 488.784,Z 279.336,A -85,B 0,C 180,E1 22870.132,E2 22870.132} C_VEL
LIN {X 0,Y 488.832,Z 279.346,A -85,B 0,C 180,E1 22866.695,E2 22866.695} C_VEL
LIN {X 0,Y 488.807,Z 279.326,A -85,B 0,C 180,E1 22863.166,E2 22863.166} C_VEL
LIN {X 0,Y 488.786,Z 279.347,A -85,B 0,C 180,E1 22859.648,E2 22859.648} C_VEL
LIN {X 0,Y 488.8,Z 279.327,A -85,B 0,C 180,E1 22856.129,E2 22856.129} C_VEL
LIN {X 0,Y 488.835,Z 279.339,A -85,B 0,C 180,E1 22852.596,E2 22852.596} C_VEL
LIN {X 0,Y 488.809,Z 279.334,A -85,B 0,C 180,E1 22849.034,E2 22849.034} C_VEL
LIN {X 0,Y 488.79,Z 279.339,A -85,B 0,C 180,E1 22845.549,E2 22845.549} C_VEL
LIN {X 0,Y 488.814,Z 279.344,A -85,B 0,C 180,E1 22842.009,E2 22842.009} C_VEL
LIN {X 0,Y 488.836,Z 279.346,A -85,B 0,C 180,E1 22838.397,E2 22838.397} C_VEL
LIN {X 0,Y 488.817,Z 279.349,A -85,B 0,C 180,E1 22834.821,E2 22834.821} C_VEL
LIN {X 0,Y 488.798,Z 279.348,A -85,B 0,C 180,E1 22831.269,E2 22831.269} C_VEL
LIN {X 0,Y 488.814,Z 279.344,A -85,B 0,C 180,E1 22827.733,E2 22827.733} C_VEL
LIN {X 0,Y 488.832,Z 279.345,A -85,B 0,C 180,E1 22824.198,E2 22824.198} C_VEL
LIN {X 0,Y 488.825,Z 279.345,A -85,B 0,C 180,E1 22820.638,E2 22820.638} C_VEL
LIN {X 0,Y 488.804,Z 279.347,A -85,B 0,C 180,E1 22817.066,E2 22817.066} C_VEL
LIN {X 0,Y 488.814,Z 279.344,A -85,B 0,C 180,E1 22813.436,E2 22813.436} C_VEL
LIN {X 0,Y 488.831,Z 279.345,A -85,B 0,C 180,E1 22809.912,E2 22809.912} C_VEL
LIN {X 0,Y 488.829,Z 279.346,A -85,B 0,C 180,E1 22806.304,E2 22806.304} C_VEL
LIN {X 0,Y 488.812,Z 279.345,A -85,B 0,C 180,E1 22802.787,E2 22802.787} C_VEL
LIN {X 0,Y 488.828,Z 279.346,A -85,B 0,C 180,E1 22802.058,E2 22802.058} C_VEL
LIN {X 0,Y 487.838,Z 279.465,A -85,B 0,C 180,E1 22801.155,E2 22801.155} C_VEL
LIN {X 0,Y 481.324,Z 280.283,A -85,B 0,C 180,E1 22798.55,E2 22798.55} C_VEL
LIN {X 0,Y 480.889,Z 280.333,A -85,B 0,C 180,E1 22797.954,E2 22797.954} C_VEL
LIN {X 0,Y 480.887,Z 280.337,A -85,B 0,C 180,E1 22794.31,E2 22794.31} C_VEL
LIN {X 0,Y 480.874,Z 280.335,A -85,B 0,C 180,E1 22790.699,E2 22790.699} C_VEL
LIN {X 0,Y 480.882,Z 280.333,A -85,B 0,C 180,E1 22787.047,E2 22787.047} C_VEL
LIN {X 0,Y 480.887,Z 280.334,A -85,B 0,C 180,E1 22783.466,E2 22783.466} C_VEL
LIN {X 0,Y 480.884,Z 280.336,A -85,B 0,C 180,E1 22779.816,E2 22779.816} C_VEL
LIN {X 0,Y 480.887,Z 280.333,A -85,B 0,C 180,E1 22776.207,E2 22776.207} C_VEL
LIN {X 0,Y 480.88,Z 280.332,A -85,B 0,C 180,E1 22772.622,E2 22772.622} C_VEL
LIN {X 0,Y 480.889,Z 280.329,A -85,B 0,C 180,E1 22769.047,E2 22769.047} C_VEL
LIN {X 0,Y 480.879,Z 280.333,A -85,B 0,C 180,E1 22765.468,E2 22765.468} C_VEL
LIN {X 0,Y 480.891,Z 280.333,A -85,B 0,C 180,E1 22761.872,E2 22761.872} C_VEL
LIN {X 0,Y 480.885,Z 280.335,A -85,B 0,C 180,E1 22758.243,E2 22758.243} C_VEL
LIN {X 0,Y 480.891,Z 280.333,A -85,B 0,C 180,E1 22754.566,E2 22754.566} C_VEL
LIN {X 0,Y 480.881,Z 280.333,A -85,B 0,C 180,E1 22750.948,E2 22750.948} C_VEL
LIN {X 0,Y 480.875,Z 280.336,A -85,B 0,C 180,E1 22747.378,E2 22747.378} C_VEL
LIN {X 0,Y 480.891,Z 280.335,A -85,B 0,C 180,E1 22743.847,E2 22743.847} C_VEL
LIN {X 0,Y 480.888,Z 280.332,A -85,B 0,C 180,E1 22740.204,E2 22740.204} C_VEL
LIN {X 0,Y 480.886,Z 280.331,A -85,B 0,C 180,E1 22736.566,E2 22736.566} C_VEL
LIN {X 0,Y 480.869,Z 280.335,A -85,B 0,C 180,E1 22732.917,E2 22732.917} C_VEL
LIN {X 0,Y 480.879,Z 280.334,A -85,B 0,C 180,E1 22729.369,E2 22729.369} C_VEL
LIN {X 0,Y 480.891,Z 280.335,A -85,B 0,C 180,E1 22725.833,E2 22725.833} C_VEL
LIN {X 0,Y 480.889,Z 280.333,A -85,B 0,C 180,E1 22722.189,E2 22722.189} C_VEL
LIN {X 0,Y 480.867,Z 280.335,A -85,B 0,C 180,E1 22718.575,E2 22718.575} C_VEL
LIN {X 0,Y 480.866,Z 280.338,A -85,B 0,C 180,E1 22714.994,E2 22714.994} C_VEL
LIN {X 0,Y 480.894,Z 280.333,A -85,B 0,C 180,E1 22711.458,E2 22711.458} C_VEL
LIN {X 0,Y 480.896,Z 280.333,A -85,B 0,C 180,E1 22707.892,E2 22707.892} C_VEL
LIN {X 0,Y 480.865,Z 280.334,A -85,B 0,C 180,E1 22704.312,E2 22704.312} C_VEL
LIN {X 0,Y 480.856,Z 280.336,A -85,B 0,C 180,E1 22700.663,E2 22700.663} C_VEL
LIN {X 0,Y 480.882,Z 280.326,A -85,B 0,C 180,E1 22697.172,E2 22697.172} C_VEL
LIN {X 0,Y 480.896,Z 280.326,A -85,B 0,C 180,E1 22693.588,E2 22693.588} C_VEL
LIN {X 0,Y 480.859,Z 280.315,A -85,B 0,C 180,E1 22690.059,E2 22690.059} C_VEL
LIN {X 0,Y 480.85,Z 280.336,A -85,B 0,C 180,E1 22686.447,E2 22686.447} C_VEL
LIN {X 0,Y 480.866,Z 280.315,A -85,B 0,C 180,E1 22682.86,E2 22682.86} C_VEL
LIN {X 0,Y 480.898,Z 280.329,A -85,B 0,C 180,E1 22679.285,E2 22679.285} C_VEL
LIN {X 0,Y 480.862,Z 280.324,A -85,B 0,C 180,E1 22675.707,E2 22675.707} C_VEL
LIN {X 0,Y 480.842,Z 280.324,A -85,B 0,C 180,E1 22672.232,E2 22672.232} C_VEL
LIN {X 0,Y 480.866,Z 280.336,A -85,B 0,C 180,E1 22668.729,E2 22668.729} C_VEL
LIN {X 0,Y 480.892,Z 280.311,A -85,B 0,C 180,E1 22665.183,E2 22665.183} C_VEL
LIN {X 0,Y 480.847,Z 280.336,A -85,B 0,C 180,E1 22661.701,E2 22661.701} C_VEL
LIN {X 0,Y 480.835,Z 280.333,A -85,B 0,C 180,E1 22658.148,E2 22658.148} C_VEL
LIN {X 0,Y 480.878,Z 280.317,A -85,B 0,C 180,E1 22654.748,E2 22654.748} C_VEL
LIN {X 0,Y 480.875,Z 280.336,A -85,B 0,C 180,E1 22651.159,E2 22651.159} C_VEL
LIN {X 0,Y 480.833,Z 280.339,A -85,B 0,C 180,E1 22647.696,E2 22647.696} C_VEL
LIN {X 0,Y 480.836,Z 280.338,A -85,B 0,C 180,E1 22644.099,E2 22644.099} C_VEL
LIN {X 0,Y 480.881,Z 280.291,A -85,B 0,C 180,E1 22640.642,E2 22640.642} C_VEL
LIN {X 0,Y 480.838,Z 280.306,A -85,B 0,C 180,E1 22637.224,E2 22637.224} C_VEL
LIN {X 0,Y 480.868,Z 280.606,A -85,B 0,C 180,E1 22635.889,E2 22635.889} C_VEL
LIN {X 0,Y 486.303,Z 296.08,A -85,B 0,C 180,E1 22632.95,E2 22632.95} C_VEL
LIN {X 0,Y 488.809,Z 303.372,A -85,B 0,C 180,E1 22631.703,E2 22631.703} C_VEL
LIN {X 0,Y 498.693,Z 320.784,A -85,B 0,C 180,E1 22630.37,E2 22630.37} C_VEL
LIN {X 0,Y 503.389,Z 338.002,A -85,B 0,C 180,E1 22629.608,E2 22629.608} C_VEL
LIN {X 0,Y 499.534,Z 552.607,A -85,B 0,C 180,E1 22626.145,E2 22626.145} C_VEL
LIN {X 0,Y 498.451,Z 608.011,A -85,B 0,C 180,E1 22625.229,E2 22625.229} C_VEL
LIN {X 0,Y 497.406,Z 631.15,A -85,B 0,C 180,E1 22624.64,E2 22624.64} C_VEL
LIN {X 0,Y 496.304,Z 649.671,A -85,B 0,C 180,E1 22623.989,E2 22623.989} C_VEL
LIN {X 0,Y 494.981,Z 668.643,A -85,B 0,C 180,E1 22623.154,E2 22623.154} C_VEL
LIN {X 0,Y 493.309,Z 689.533,A -85,B 0,C 180,E1 22622.006,E2 22622.006} C_VEL
LIN {X 0,Y 491.748,Z 706.704,A -85,B 0,C 180,E1 22620.87,E2 22620.87} C_VEL
LIN {X 0,Y 490.226,Z 722.674,A -85,B 0,C 180,E1 22619.642,E2 22619.642} C_VEL
LIN {X 0,Y 488.298,Z 741.928,A -85,B 0,C 180,E1 22617.899,E2 22617.899} C_VEL
LIN {X 0,Y 486.688,Z 757.415,A -85,B 0,C 180,E1 22616.251,E2 22616.251} C_VEL
LIN {X 0,Y 485.15,Z 772.889,A -85,B 0,C 180,E1 22614.366,E2 22614.366} C_VEL
LIN {X 0,Y 483.687,Z 787.827,A -85,B 0,C 180,E1 22612.227,E2 22612.227} C_VEL
LIN {X 0,Y 482.611,Z 799.84,A -85,B 0,C 180,E1 22610.241,E2 22610.241} C_VEL
LIN {X 0,Y 481.636,Z 812.126,A -85,B 0,C 180,E1 22607.893,E2 22607.893} C_VEL
LIN {X 0,Y 480.93,Z 822.331,A -85,B 0,C 180,E1 22605.556,E2 22605.556} C_VEL
LIN {X 0,Y 480.465,Z 830.913,A -85,B 0,C 180,E1 22603.233,E2 22603.233} C_VEL
LIN {X 0,Y 480.149,Z 838.832,A -85,B 0,C 180,E1 22600.559,E2 22600.559} C_VEL
LIN {X 0,Y 480.008,Z 844.139,A -85,B 0,C 180,E1 22598.263,E2 22598.263} C_VEL
LIN {X 0,Y 479.934,Z 848.511,A -85,B 0,C 180,E1 22595.739,E2 22595.739} C_VEL
LIN {X 0,Y 479.915,Z 851.279,A -85,B 0,C 180,E1 22593.105,E2 22593.105} C_VEL
LIN {X 0,Y 479.905,Z 852.337,A -85,B 0,C 180,E1 22590.836,E2 22590.836} C_VEL
LIN {X 0,Y 479.898,Z 852.176,A -85,B 0,C 180,E1 22588.448,E2 22588.448} C_VEL
LIN {X 0,Y 479.916,Z 850.351,A -85,B 0,C 180,E1 22585.818,E2 22585.818} C_VEL
LIN {X 0,Y 479.942,Z 847.194,A -85,B 0,C 180,E1 22583.421,E2 22583.421} C_VEL
LIN {X 0,Y 480.032,Z 842.652,A -85,B 0,C 180,E1 22581.013,E2 22581.013} C_VEL
LIN {X 0,Y 480.254,Z 835.823,A -85,B 0,C 180,E1 22578.349,E2 22578.349} C_VEL
LIN {X 0,Y 480.596,Z 828.359,A -85,B 0,C 180,E1 22576.035,E2 22576.035} C_VEL
LIN {X 0,Y 481.206,Z 818.294,A -85,B 0,C 180,E1 22573.462,E2 22573.462} C_VEL
LIN {X 0,Y 482.013,Z 807.162,A -85,B 0,C 180,E1 22571.12,E2 22571.12} C_VEL
LIN {X 0,Y 483.058,Z 794.874,A -85,B 0,C 180,E1 22568.891,E2 22568.891} C_VEL
LIN {X 0,Y 484.407,Z 780.258,A -85,B 0,C 180,E1 22566.653,E2 22566.653} C_VEL
LIN {X 0,Y 485.75,Z 766.672,A -85,B 0,C 180,E1 22564.847,E2 22564.847} C_VEL
LIN {X 0,Y 487.519,Z 749.611,A -85,B 0,C 180,E1 22562.885,E2 22562.885} C_VEL
LIN {X 0,Y 489.142,Z 733.371,A -85,B 0,C 180,E1 22561.292,E2 22561.292} C_VEL
LIN {X 0,Y 490.77,Z 717.308,A -85,B 0,C 180,E1 22559.923,E2 22559.923} C_VEL
LIN {X 0,Y 492.679,Z 696.451,A -85,B 0,C 180,E1 22558.427,E2 22558.427} C_VEL
LIN {X 0,Y 494.18,Z 678.707,A -85,B 0,C 180,E1 22557.372,E2 22557.372} C_VEL
LIN {X 0,Y 495.581,Z 660.722,A -85,B 0,C 180,E1 22556.476,E2 22556.476} C_VEL
LIN {X 0,Y 497.034,Z 637.539,A -85,B 0,C 180,E1 22555.564,E2 22555.564} C_VEL
LIN {X 0,Y 497.991,Z 618.68,A -85,B 0,C 180,E1 22555.015,E2 22555.015} C_VEL
LIN {X 0,Y 498.754,Z 597.999,A -85,B 0,C 180,E1 22554.584,E2 22554.584} C_VEL
LIN {X 0,Y 502.687,Z 375.938,A -85,B 0,C 180,E1 22551.01,E2 22551.01} C_VEL
LIN {X 0,Y 503.231,Z 336.781,A -85,B 0,C 180,E1 22550.355,E2 22550.355} C_VEL
LIN {X 0,Y 498.131,Z 319.452,A -85,B 0,C 180,E1 22549.551,E2 22549.551} C_VEL
LIN {X 0,Y 488.581,Z 302.868,A -85,B 0,C 180,E1 22548.239,E2 22548.239} C_VEL
LIN {X 0,Y 483.645,Z 288.605,A -85,B 0,C 180,E1 22545.667,E2 22545.667} C_VEL
LIN {X 0,Y 480.847,Z 280.461,A -85,B 0,C 180,E1 22544.062,E2 22544.062} C_VEL
LIN {X 0,Y 480.826,Z 280.324,A -85,B 0,C 180,E1 22540.442,E2 22540.442} C_VEL
LIN {X 0,Y 480.871,Z 280.309,A -85,B 0,C 180,E1 22537.021,E2 22537.021} C_VEL
LIN {X 0,Y 480.862,Z 280.327,A -85,B 0,C 180,E1 22533.511,E2 22533.511} C_VEL
LIN {X 0,Y 480.83,Z 280.326,A -85,B 0,C 180,E1 22530.076,E2 22530.076} C_VEL
LIN {X 0,Y 480.849,Z 280.323,A -85,B 0,C 180,E1 22526.555,E2 22526.555} C_VEL
LIN {X 0,Y 480.896,Z 280.332,A -85,B 0,C 180,E1 22523.009,E2 22523.009} C_VEL
LIN {X 0,Y 480.858,Z 280.32,A -85,B 0,C 180,E1 22519.432,E2 22519.432} C_VEL
LIN {X 0,Y 480.838,Z 280.325,A -85,B 0,C 180,E1 22515.931,E2 22515.931} C_VEL
LIN {X 0,Y 480.858,Z 280.334,A -85,B 0,C 180,E1 22512.367,E2 22512.367} C_VEL
LIN {X 0,Y 480.891,Z 280.31,A -85,B 0,C 180,E1 22508.851,E2 22508.851} C_VEL
LIN {X 0,Y 480.857,Z 280.339,A -85,B 0,C 180,E1 22505.369,E2 22505.369} C_VEL
LIN {X 0,Y 480.844,Z 280.322,A -85,B 0,C 180,E1 22501.787,E2 22501.787} C_VEL
LIN {X 0,Y 480.875,Z 280.325,A -85,B 0,C 180,E1 22498.332,E2 22498.332} C_VEL
LIN {X 0,Y 480.889,Z 280.326,A -85,B 0,C 180,E1 22494.751,E2 22494.751} C_VEL
LIN {X 0,Y 480.857,Z 280.32,A -85,B 0,C 180,E1 22491.269,E2 22491.269} C_VEL
LIN {X 0,Y 480.851,Z 280.335,A -85,B 0,C 180,E1 22487.633,E2 22487.633} C_VEL
LIN {X 0,Y 480.875,Z 280.314,A -85,B 0,C 180,E1 22484.07,E2 22484.07} C_VEL
LIN {X 0,Y 480.894,Z 280.334,A -85,B 0,C 180,E1 22480.443,E2 22480.443} C_VEL
LIN {X 0,Y 480.878,Z 280.337,A -85,B 0,C 180,E1 22476.86,E2 22476.86} C_VEL
LIN {X 0,Y 480.859,Z 280.336,A -85,B 0,C 180,E1 22473.312,E2 22473.312} C_VEL
LIN {X 0,Y 480.877,Z 280.333,A -85,B 0,C 180,E1 22469.79,E2 22469.79} C_VEL
LIN {X 0,Y 480.894,Z 280.334,A -85,B 0,C 180,E1 22466.268,E2 22466.268} C_VEL
LIN {X 0,Y 480.887,Z 280.334,A -85,B 0,C 180,E1 22462.583,E2 22462.583} C_VEL
LIN {X 0,Y 480.866,Z 280.337,A -85,B 0,C 180,E1 22459.004,E2 22459.004} C_VEL
LIN {X 0,Y 480.869,Z 280.334,A -85,B 0,C 180,E1 22455.324,E2 22455.324} C_VEL
LIN {X 0,Y 480.894,Z 280.332,A -85,B 0,C 180,E1 22451.706,E2 22451.706} C_VEL
LIN {X 0,Y 480.892,Z 280.336,A -85,B 0,C 180,E1 22448.134,E2 22448.134} C_VEL
LIN {X 0,Y 480.879,Z 280.334,A -85,B 0,C 180,E1 22444.576,E2 22444.576} C_VEL
LIN {X 0,Y 480.872,Z 280.333,A -85,B 0,C 180,E1 22441.04,E2 22441.04} C_VEL
LIN {X 0,Y 480.889,Z 280.333,A -85,B 0,C 180,E1 22437.954,E2 22437.954} C_VEL
LIN {X 0,Y 479.901,Z 280.453,A -85,B 0,C 180,E1 22437.036,E2 22437.036} C_VEL
LIN {X 0,Y 473.387,Z 281.272,A -85,B 0,C 180,E1 22434.388,E2 22434.388} C_VEL
LIN {X 0,Y 472.95,Z 281.32,A -85,B 0,C 180,E1 22433.782,E2 22433.782} C_VEL
LIN {X 0,Y 472.952,Z 281.322,A -85,B 0,C 180,E1 22430.156,E2 22430.156} C_VEL
LIN {X 0,Y 472.943,Z 281.325,A -85,B 0,C 180,E1 22426.456,E2 22426.456} C_VEL
LIN {X 0,Y 472.94,Z 281.324,A -85,B 0,C 180,E1 22422.825,E2 22422.825} C_VEL
LIN {X 0,Y 472.951,Z 281.321,A -85,B 0,C 180,E1 22419.123,E2 22419.123} C_VEL
LIN {X 0,Y 472.942,Z 281.324,A -85,B 0,C 180,E1 22415.581,E2 22415.581} C_VEL
LIN {X 0,Y 472.949,Z 281.326,A -85,B 0,C 180,E1 22411.938,E2 22411.938} C_VEL
LIN {X 0,Y 472.945,Z 281.323,A -85,B 0,C 180,E1 22408.304,E2 22408.304} C_VEL
LIN {X 0,Y 472.945,Z 281.322,A -85,B 0,C 180,E1 22404.663,E2 22404.663} C_VEL
LIN {X 0,Y 472.944,Z 281.323,A -85,B 0,C 180,E1 22401.122,E2 22401.122} C_VEL
LIN {X 0,Y 472.938,Z 281.325,A -85,B 0,C 180,E1 22397.423,E2 22397.423} C_VEL
LIN {X 0,Y 472.95,Z 281.322,A -85,B 0,C 180,E1 22393.796,E2 22393.796} C_VEL
LIN {X 0,Y 472.947,Z 281.321,A -85,B 0,C 180,E1 22390.101,E2 22390.101} C_VEL
LIN {X 0,Y 472.952,Z 281.319,A -85,B 0,C 180,E1 22386.45,E2 22386.45} C_VEL
LIN {X 0,Y 472.94,Z 281.319,A -85,B 0,C 180,E1 22382.83,E2 22382.83} C_VEL
LIN {X 0,Y 472.933,Z 281.322,A -85,B 0,C 180,E1 22379.229,E2 22379.229} C_VEL
LIN {X 0,Y 472.95,Z 281.323,A -85,B 0,C 180,E1 22375.636,E2 22375.636} C_VEL
LIN {X 0,Y 472.952,Z 281.323,A -85,B 0,C 180,E1 22372.035,E2 22372.035} C_VEL
LIN {X 0,Y 472.949,Z 281.322,A -85,B 0,C 180,E1 22368.409,E2 22368.409} C_VEL
LIN {X 0,Y 472.929,Z 281.324,A -85,B 0,C 180,E1 22364.737,E2 22364.737} C_VEL
LIN {X 0,Y 472.931,Z 281.326,A -85,B 0,C 180,E1 22361.11,E2 22361.11} C_VEL
LIN {X 0,Y 472.951,Z 281.322,A -85,B 0,C 180,E1 22357.507,E2 22357.507} C_VEL
LIN {X 0,Y 472.956,Z 281.323,A -85,B 0,C 180,E1 22353.819,E2 22353.819} C_VEL
LIN {X 0,Y 472.942,Z 281.322,A -85,B 0,C 180,E1 22350.157,E2 22350.157} C_VEL
LIN {X 0,Y 472.92,Z 281.324,A -85,B 0,C 180,E1 22346.583,E2 22346.583} C_VEL
LIN {X 0,Y 472.926,Z 281.326,A -85,B 0,C 180,E1 22342.893,E2 22342.893} C_VEL
LIN {X 0,Y 472.953,Z 281.325,A -85,B 0,C 180,E1 22339.385,E2 22339.385} C_VEL
LIN {X 0,Y 472.95,Z 281.299,A -85,B 0,C 180,E1 22335.7,E2 22335.7} C_VEL
LIN {X 0,Y 472.916,Z 281.324,A -85,B 0,C 180,E1 22332.206,E2 22332.206} C_VEL
LIN {X 0,Y 472.911,Z 281.312,A -85,B 0,C 180,E1 22328.511,E2 22328.511} C_VEL
LIN {X 0,Y 472.936,Z 281.311,A -85,B 0,C 180,E1 22324.973,E2 22324.973} C_VEL
LIN {X 0,Y 472.955,Z 281.315,A -85,B 0,C 180,E1 22321.333,E2 22321.333} C_VEL
LIN {X 0,Y 472.919,Z 281.304,A -85,B 0,C 180,E1 22317.819,E2 22317.819} C_VEL
LIN {X 0,Y 472.906,Z 281.326,A -85,B 0,C 180,E1 22314.175,E2 22314.175} C_VEL
LIN {X 0,Y 472.918,Z 281.303,A -85,B 0,C 180,E1 22310.631,E2 22310.631} C_VEL
LIN {X 0,Y 472.952,Z 281.318,A -85,B 0,C 180,E1 22307.049,E2 22307.049} C_VEL
LIN {X 0,Y 472.919,Z 281.316,A -85,B 0,C 180,E1 22303.542,E2 22303.542} C_VEL
LIN {X 0,Y 472.896,Z 281.307,A -85,B 0,C 180,E1 22299.969,E2 22299.969} C_VEL
LIN {X 0,Y 472.914,Z 281.325,A -85,B 0,C 180,E1 22296.447,E2 22296.447} C_VEL
LIN {X 0,Y 472.949,Z 281.313,A -85,B 0,C 180,E1 22292.829,E2 22292.829} C_VEL
LIN {X 0,Y 472.911,Z 281.313,A -85,B 0,C 180,E1 22289.367,E2 22289.367} C_VEL
LIN {X 0,Y 472.89,Z 281.32,A -85,B 0,C 180,E1 22285.777,E2 22285.777} C_VEL
LIN {X 0,Y 472.897,Z 281.283,A -85,B 0,C 180,E1 22282.182,E2 22282.182} C_VEL
LIN {X 0,Y 472.948,Z 281.326,A -85,B 0,C 180,E1 22278.632,E2 22278.632} C_VEL
LIN {X 0,Y 472.976,Z 281.562,A -85,B 0,C 180,E1 22276.663,E2 22276.663} C_VEL
LIN {X 0,Y 478.574,Z 297.538,A -85,B 0,C 180,E1 22273.534,E2 22273.534} C_VEL
LIN {X 0,Y 480.463,Z 303.01,A -85,B 0,C 180,E1 22272.594,E2 22272.594} C_VEL
LIN {X 0,Y 493.165,Z 325.032,A -85,B 0,C 180,E1 22270.834,E2 22270.834} C_VEL
LIN {X 0,Y 497.172,Z 340.108,A -85,B 0,C 180,E1 22270.16,E2 22270.16} C_VEL
LIN {X 0,Y 493.025,Z 554.653,A -85,B 0,C 180,E1 22266.658,E2 22266.658} C_VEL
LIN {X 0,Y 491.899,Z 607.949,A -85,B 0,C 180,E1 22265.766,E2 22265.766} C_VEL
LIN {X 0,Y 490.784,Z 631.019,A -85,B 0,C 180,E1 22265.171,E2 22265.171} C_VEL
LIN {X 0,Y 489.614,Z 649.419,A -85,B 0,C 180,E1 22264.519,E2 22264.519} C_VEL
LIN {X 0,Y 488.192,Z 668.391,A -85,B 0,C 180,E1 22263.677,E2 22263.677} C_VEL
LIN {X 0,Y 486.4,Z 689.279,A -85,B 0,C 180,E1 22262.516,E2 22262.516} C_VEL
LIN {X 0,Y 484.698,Z 706.712,A -85,B 0,C 180,E1 22261.349,E2 22261.349} C_VEL
LIN {X 0,Y 482.939,Z 724.003,A -85,B 0,C 180,E1 22259.999,E2 22259.999} C_VEL
LIN {X 0,Y 480.895,Z 743.139,A -85,B 0,C 180,E1 22258.229,E2 22258.229} C_VEL
LIN {X 0,Y 479.327,Z 757.195,A -85,B 0,C 180,E1 22256.712,E2 22256.712} C_VEL
LIN {X 0,Y 477.772,Z 771.592,A -85,B 0,C 180,E1 22254.941,E2 22254.941} C_VEL
LIN {X 0,Y 476.14,Z 787.029,A -85,B 0,C 180,E1 22252.729,E2 22252.729} C_VEL
LIN {X 0,Y 474.941,Z 799.128,A -85,B 0,C 180,E1 22250.712,E2 22250.712} C_VEL
LIN {X 0,Y 473.92,Z 810.948,A -85,B 0,C 180,E1 22248.449,E2 22248.449} C_VEL
LIN {X 0,Y 473.071,Z 821.955,A -85,B 0,C 180,E1 22245.917,E2 22245.917} C_VEL
LIN {X 0,Y 472.55,Z 830.483,A -85,B 0,C 180,E1 22243.583,E2 22243.583} C_VEL
LIN {X 0,Y 472.181,Z 838.526,A -85,B 0,C 180,E1 22240.863,E2 22240.863} C_VEL
LIN {X 0,Y 472.012,Z 843.89,A -85,B 0,C 180,E1 22238.527,E2 22238.527} C_VEL
LIN {X 0,Y 471.939,Z 848.141,A -85,B 0,C 180,E1 22236.081,E2 22236.081} C_VEL
LIN {X 0,Y 471.915,Z 851.195,A -85,B 0,C 180,E1 22233.279,E2 22233.279} C_VEL
LIN {X 0,Y 471.91,Z 852.308,A -85,B 0,C 180,E1 22230.971,E2 22230.971} C_VEL
LIN {X 0,Y 471.904,Z 852.228,A -85,B 0,C 180,E1 22228.665,E2 22228.665} C_VEL
LIN {X 0,Y 471.912,Z 850.608,A -85,B 0,C 180,E1 22225.991,E2 22225.991} C_VEL
LIN {X 0,Y 471.94,Z 847.531,A -85,B 0,C 180,E1 22223.528,E2 22223.528} C_VEL
LIN {X 0,Y 472.018,Z 843.397,A -85,B 0,C 180,E1 22221.228,E2 22221.228} C_VEL
LIN {X 0,Y 472.24,Z 837.146,A -85,B 0,C 180,E1 22218.606,E2 22218.606} C_VEL
LIN {X 0,Y 472.597,Z 829.632,A -85,B 0,C 180,E1 22216.169,E2 22216.169} C_VEL
LIN {X 0,Y 473.159,Z 820.854,A -85,B 0,C 180,E1 22213.804,E2 22213.804} C_VEL
LIN {X 0,Y 474.069,Z 809.053,A -85,B 0,C 180,E1 22211.175,E2 22211.175} C_VEL
LIN {X 0,Y 475.006,Z 798.417,A -85,B 0,C 180,E1 22209.162,E2 22209.162} C_VEL
LIN {X 0,Y 476.311,Z 785.442,A -85,B 0,C 180,E1 22207.018,E2 22207.018} C_VEL
LIN {X 0,Y 477.921,Z 770.114,A -85,B 0,C 180,E1 22204.869,E2 22204.869} C_VEL
LIN {X 0,Y 479.403,Z 756.505,A -85,B 0,C 180,E1 22203.208,E2 22203.208} C_VEL
LIN {X 0,Y 481.19,Z 740.632,A -85,B 0,C 180,E1 22201.515,E2 22201.515} C_VEL
LIN {X 0,Y 483.054,Z 722.836,A -85,B 0,C 180,E1 22199.906,E2 22199.906} C_VEL
LIN {X 0,Y 484.75,Z 706.2,A -85,B 0,C 180,E1 22198.614,E2 22198.614} C_VEL
LIN {X 0,Y 486.504,Z 688.236,A -85,B 0,C 180,E1 22197.418,E2 22197.418} C_VEL
LIN {X 0,Y 488.289,Z 667.07,A -85,B 0,C 180,E1 22196.261,E2 22196.261} C_VEL
LIN {X 0,Y 489.614,Z 649.419,A -85,B 0,C 180,E1 22195.481,E2 22195.481} C_VEL
LIN {X 0,Y 490.786,Z 631.019,A -85,B 0,C 180,E1 22194.829,E2 22194.829} C_VEL
LIN {X 0,Y 491.899,Z 607.949,A -85,B 0,C 180,E1 22194.234,E2 22194.234} C_VEL
LIN {X 0,Y 493.042,Z 553.76,A -85,B 0,C 180,E1 22193.327,E2 22193.327} C_VEL
LIN {X 0,Y 497.185,Z 339.493,A -85,B 0,C 180,E1 22189.83,E2 22189.83} C_VEL
LIN {X 0,Y 492.641,Z 323.886,A -85,B 0,C 180,E1 22189.092,E2 22189.092} C_VEL
LIN {X 0,Y 480.241,Z 302.47,A -85,B 0,C 180,E1 22187.346,E2 22187.346} C_VEL
LIN {X 0,Y 474.851,Z 287.08,A -85,B 0,C 180,E1 22184.456,E2 22184.456} C_VEL
LIN {X 0,Y 472.954,Z 281.412,A -85,B 0,C 180,E1 22183.267,E2 22183.267} C_VEL
LIN {X 0,Y 472.897,Z 281.292,A -85,B 0,C 180,E1 22179.84,E2 22179.84} C_VEL
LIN {X 0,Y 472.891,Z 281.323,A -85,B 0,C 180,E1 22176.3,E2 22176.3} C_VEL
LIN {X 0,Y 472.918,Z 281.324,A -85,B 0,C 180,E1 22172.768,E2 22172.768} C_VEL
LIN {X 0,Y 472.953,Z 281.315,A -85,B 0,C 180,E1 22169.18,E2 22169.18} C_VEL
LIN {X 0,Y 472.905,Z 281.306,A -85,B 0,C 180,E1 22165.685,E2 22165.685} C_VEL
LIN {X 0,Y 472.897,Z 281.322,A -85,B 0,C 180,E1 22162.108,E2 22162.108} C_VEL
LIN {X 0,Y 472.928,Z 281.323,A -85,B 0,C 180,E1 22158.617,E2 22158.617} C_VEL
LIN {X 0,Y 472.947,Z 281.297,A -85,B 0,C 180,E1 22155.072,E2 22155.072} C_VEL
LIN {X 0,Y 472.909,Z 281.326,A -85,B 0,C 180,E1 22151.587,E2 22151.587} C_VEL
LIN {X 0,Y 472.905,Z 281.312,A -85,B 0,C 180,E1 22148.021,E2 22148.021} C_VEL
LIN {X 0,Y 472.937,Z 281.313,A -85,B 0,C 180,E1 22144.486,E2 22144.486} C_VEL
LIN {X 0,Y 472.953,Z 281.315,A -85,B 0,C 180,E1 22140.848,E2 22140.848} C_VEL
LIN {X 0,Y 472.916,Z 281.306,A -85,B 0,C 180,E1 22137.334,E2 22137.334} C_VEL
LIN {X 0,Y 472.911,Z 281.325,A -85,B 0,C 180,E1 22133.688,E2 22133.688} C_VEL
LIN {X 0,Y 472.931,Z 281.3,A -85,B 0,C 180,E1 22130.123,E2 22130.123} C_VEL
LIN {X 0,Y 472.958,Z 281.316,A -85,B 0,C 180,E1 22126.517,E2 22126.517} C_VEL
LIN {X 0,Y 472.941,Z 281.314,A -85,B 0,C 180,E1 22122.854,E2 22122.854} C_VEL
LIN {X 0,Y 472.919,Z 281.325,A -85,B 0,C 180,E1 22119.324,E2 22119.324} C_VEL
LIN {X 0,Y 472.925,Z 281.323,A -85,B 0,C 180,E1 22115.653,E2 22115.653} C_VEL
LIN {X 0,Y 472.951,Z 281.322,A -85,B 0,C 180,E1 22112.01,E2 22112.01} C_VEL
LIN {X 0,Y 472.955,Z 281.322,A -85,B 0,C 180,E1 22108.38,E2 22108.38} C_VEL
LIN {X 0,Y 472.944,Z 281.323,A -85,B 0,C 180,E1 22104.689,E2 22104.689} C_VEL
LIN {X 0,Y 472.926,Z 281.326,A -85,B 0,C 180,E1 22101.078,E2 22101.078} C_VEL
LIN {X 0,Y 472.932,Z 281.323,A -85,B 0,C 180,E1 22097.427,E2 22097.427} C_VEL
LIN {X 0,Y 472.952,Z 281.322,A -85,B 0,C 180,E1 22093.871,E2 22093.871} C_VEL
LIN {X 0,Y 472.955,Z 281.323,A -85,B 0,C 180,E1 22090.255,E2 22090.255} C_VEL
LIN {X 0,Y 472.94,Z 281.323,A -85,B 0,C 180,E1 22086.596,E2 22086.596} C_VEL
LIN {X 0,Y 472.933,Z 281.322,A -85,B 0,C 180,E1 22082.91,E2 22082.91} C_VEL
LIN {X 0,Y 472.942,Z 281.32,A -85,B 0,C 180,E1 22079.232,E2 22079.232} C_VEL
LIN {X 0,Y 472.95,Z 281.319,A -85,B 0,C 180,E1 22075.682,E2 22075.682} C_VEL
LIN {X 0,Y 472.95,Z 281.32,A -85,B 0,C 180,E1 22073.782,E2 22073.782} C_VEL
LIN {X 0,Y 471.961,Z 281.445,A -85,B 0,C 180,E1 22072.849,E2 22072.849} C_VEL
LIN {X 0,Y 465.443,Z 282.258,A -85,B 0,C 180,E1 22070.156,E2 22070.156} C_VEL
LIN {X 0,Y 465.011,Z 282.31,A -85,B 0,C 180,E1 22069.539,E2 22069.539} C_VEL
LIN {X 0,Y 465.01,Z 282.31,A -85,B 0,C 180,E1 22065.847,E2 22065.847} C_VEL
LIN {X 0,Y 465.009,Z 282.311,A -85,B 0,C 180,E1 22062.164,E2 22062.164} C_VEL
LIN {X 0,Y 465.002,Z 282.311,A -85,B 0,C 180,E1 22058.467,E2 22058.467} C_VEL
LIN {X 0,Y 465.006,Z 282.31,A -85,B 0,C 180,E1 22054.81,E2 22054.81} C_VEL
LIN {X 0,Y 465.013,Z 282.307,A -85,B 0,C 180,E1 22051.066,E2 22051.066} C_VEL
LIN {X 0,Y 465.002,Z 282.31,A -85,B 0,C 180,E1 22047.412,E2 22047.412} C_VEL
LIN {X 0,Y 465.006,Z 282.311,A -85,B 0,C 180,E1 22043.704,E2 22043.704} C_VEL
LIN {X 0,Y 465.009,Z 282.311,A -85,B 0,C 180,E1 22039.992,E2 22039.992} C_VEL
LIN {X 0,Y 465.007,Z 282.312,A -85,B 0,C 180,E1 22036.319,E2 22036.319} C_VEL
LIN {X 0,Y 465.011,Z 282.311,A -85,B 0,C 180,E1 22032.61,E2 22032.61} C_VEL
LIN {X 0,Y 465.004,Z 282.31,A -85,B 0,C 180,E1 22028.938,E2 22028.938} C_VEL
LIN {X 0,Y 464.996,Z 282.311,A -85,B 0,C 180,E1 22025.21,E2 22025.21} C_VEL
LIN {X 0,Y 465.005,Z 282.312,A -85,B 0,C 180,E1 22021.489,E2 22021.489} C_VEL
LIN {X 0,Y 465.012,Z 282.314,A -85,B 0,C 180,E1 22017.905,E2 22017.905} C_VEL
LIN {X 0,Y 465.013,Z 282.311,A -85,B 0,C 180,E1 22014.156,E2 22014.156} C_VEL
LIN {X 0,Y 465.007,Z 282.311,A -85,B 0,C 180,E1 22010.473,E2 22010.473} C_VEL
LIN {X 0,Y 464.99,Z 282.314,A -85,B 0,C 180,E1 22006.798,E2 22006.798} C_VEL
LIN {X 0,Y 464.994,Z 282.314,A -85,B 0,C 180,E1 22003.14,E2 22003.14} C_VEL
LIN {X 0,Y 465.016,Z 282.31,A -85,B 0,C 180,E1 21999.477,E2 21999.477} C_VEL
LIN {X 0,Y 465.015,Z 282.311,A -85,B 0,C 180,E1 21995.792,E2 21995.792} C_VEL
LIN {X 0,Y 465.008,Z 282.311,A -85,B 0,C 180,E1 21992.08,E2 21992.08} C_VEL
LIN {X 0,Y 464.985,Z 282.314,A -85,B 0,C 180,E1 21988.513,E2 21988.513} C_VEL
LIN {X 0,Y 464.984,Z 282.315,A -85,B 0,C 180,E1 21984.791,E2 21984.791} C_VEL
LIN {X 0,Y 465.005,Z 282.315,A -85,B 0,C 180,E1 21981.176,E2 21981.176} C_VEL
LIN {X 0,Y 465.016,Z 282.307,A -85,B 0,C 180,E1 21977.519,E2 21977.519} C_VEL
LIN {X 0,Y 465.006,Z 282.302,A -85,B 0,C 180,E1 21973.808,E2 21973.808} C_VEL
LIN {X 0,Y 464.977,Z 282.291,A -85,B 0,C 180,E1 21970.156,E2 21970.156} C_VEL
LIN {X 0,Y 464.974,Z 282.315,A -85,B 0,C 180,E1 21966.544,E2 21966.544} C_VEL
LIN {X 0,Y 464.994,Z 282.288,A -85,B 0,C 180,E1 21962.958,E2 21962.958} C_VEL
LIN {X 0,Y 465.021,Z 282.307,A -85,B 0,C 180,E1 21959.384,E2 21959.384} C_VEL
LIN {X 0,Y 464.985,Z 282.301,A -85,B 0,C 180,E1 21955.684,E2 21955.684} C_VEL
LIN {X 0,Y 464.964,Z 282.301,A -85,B 0,C 180,E1 21952.09,E2 21952.09} C_VEL
LIN {X 0,Y 464.973,Z 282.317,A -85,B 0,C 180,E1 21948.464,E2 21948.464} C_VEL
LIN {X 0,Y 465.005,Z 282.287,A -85,B 0,C 180,E1 21944.888,E2 21944.888} C_VEL
LIN {X 0,Y 464.996,Z 282.31,A -85,B 0,C 180,E1 21941.314,E2 21941.314} C_VEL
LIN {X 0,Y 464.961,Z 282.312,A -85,B 0,C 180,E1 21937.761,E2 21937.761} C_VEL
LIN {X 0,Y 464.958,Z 282.295,A -85,B 0,C 180,E1 21934.117,E2 21934.117} C_VEL
LIN {X 0,Y 464.987,Z 282.303,A -85,B 0,C 180,E1 21930.557,E2 21930.557} C_VEL
LIN {X 0,Y 465,Z 282.306,A -85,B 0,C 180,E1 21926.989,E2 21926.989} C_VEL
LIN {X 0,Y 464.958,Z 282.299,A -85,B 0,C 180,E1 21923.44,E2 21923.44} C_VEL
LIN {X 0,Y 464.947,Z 282.287,A -85,B 0,C 180,E1 21919.824,E2 21919.824} C_VEL
LIN {X 0,Y 464.991,Z 282.582,A -85,B 0,C 180,E1 21917.471,E2 21917.471} C_VEL
LIN {X 0,Y 470.448,Z 297.839,A -85,B 0,C 180,E1 21914.364,E2 21914.364} C_VEL
LIN {X 0,Y 471.983,Z 302.183,A -85,B 0,C 180,E1 21913.573,E2 21913.573} C_VEL
LIN {X 0,Y 482.997,Z 321.078,A -85,B 0,C 180,E1 21911.954,E2 21911.954} C_VEL
LIN {X 0,Y 487.792,Z 329.762,A -85,B 0,C 180,E1 21911.287,E2 21911.287} C_VEL
LIN {X 0,Y 491.002,Z 342.146,A -85,B 0,C 180,E1 21910.727,E2 21910.727} C_VEL
LIN {X 0,Y 486.575,Z 555.806,A -85,B 0,C 180,E1 21907.2,E2 21907.2} C_VEL
LIN {X 0,Y 485.392,Z 607.866,A -85,B 0,C 180,E1 21906.317,E2 21906.317} C_VEL
LIN {X 0,Y 484.205,Z 630.888,A -85,B 0,C 180,E1 21905.717,E2 21905.717} C_VEL
LIN {X 0,Y 483.029,Z 648.385,A -85,B 0,C 180,E1 21905.094,E2 21905.094} C_VEL
LIN {X 0,Y 481.6,Z 666.29,A -85,B 0,C 180,E1 21904.301,E2 21904.301} C_VEL
LIN {X 0,Y 479.733,Z 687.049,A -85,B 0,C 180,E1 21903.167,E2 21903.167} C_VEL
LIN {X 0,Y 477.862,Z 705.074,A -85,B 0,C 180,E1 21901.962,E2 21901.962} C_VEL
